METHOD SendLogMessage : BOOL
  VAR_INPUT
    str : STRING(128);
    instance : STRING(GVL_MQTT.MQTT_TOPIC_LEN) := '';
  END_VAR
                  pMqttPublishQueue^.AddMessageOn(Lane := iQueueLane,
	Payload:= CONCAT(CONCAT(instance,' | '),str),
	Topic := CONCAT(MqttDiagnosticTopic, '/Log'),
	Qos := MQTT.QoS.AtLeastOnce,
	MqttRetain := TRUE
);
                
END_METHOD

METHOD CreateSwitchEntity
  VAR_INPUT
    Name : STRING;  (* default *)
    Id : STRING;
    CommandTopic : STRING(GVL_MQTT.MQTT_TOPIC_LEN);  (* entity specific *)
    PayloadOn : STRING;
    PayloadOff : STRING;
    StateTopic : STRING(GVL_MQTT.MQTT_TOPIC_LEN);
    StateOnPayload : STRING;
    StateOffPayload : STRING;
    DeviceClass : STRING;
  END_VAR
  VAR
    EntityId : STRING(25) := 'switch';
  END_VAR
                  (* Name, id, availability and device are identical for every entity type, so
   they are filled once through the shared base struct. *)
THIS^.FillCommonFields(
	pBase := ADR(stMqttDiscMsgSwitch),
	EntityId := EntityId,
	Name := name,
	Id := Id);

// Entity related: Specific
stMqttDiscMsgSwitch.cmd_t.CharString := CommandTopic;
stMqttDiscMsgSwitch.pl_on.CharString := PayloadOn;
stMqttDiscMsgSwitch.pl_off.CharString := PayloadOff;
stMqttDiscMsgSwitch.stat_t.CharString := StateTopic;
stMqttDiscMsgSwitch.stat_on.CharString := StateOnPayload;
stMqttDiscMsgSwitch.stat_off.CharString := StateOffPayload;
stMqttDiscMsgSwitch.opt.Boolean := FALSE;
stMqttDiscMsgSwitch.dev_cla.CharString := DeviceClass;



THIS^.PublishEntityConfig(
	pStruct := ADR(stMqttDiscMsgSwitch),
	StructSize := SIZEOF(stMqttDiscMsgSwitch),
	EntityId := EntityId,
	Id := Id);
                
END_METHOD

METHOD CreateLightDimmerEntity
  VAR_INPUT
    Name : STRING;  (* default *)
    Id : STRING;
    CommandTopic : STRING(GVL_MQTT.MQTT_TOPIC_LEN);  (* entity specific *)
    PayloadOn : STRING;
    PayloadOff : STRING;
    StateTopic : STRING(GVL_MQTT.MQTT_TOPIC_LEN);
    BrightnessCommandTopic : STRING(GVL_MQTT.MQTT_TOPIC_LEN);
    BrightnessStateTopic : STRING(GVL_MQTT.MQTT_TOPIC_LEN);
    BrightnessScale : INT;
    OnCommandType : STRING := 'last';
    DmxChannel : INT := 0;  (* dmx specific *)
    DmxWidth : INT := 0;
    DmxUniverse : INT := 0;
  END_VAR
  VAR
    EntityId : STRING(25) := 'light';
  END_VAR
                  (* Name, id, availability and device are identical for every entity type, so
   they are filled once through the shared base struct. *)
THIS^.FillCommonFields(
	pBase := ADR(stMqttDiscMsgLightDim),
	EntityId := EntityId,
	Name := name,
	Id := Id);

// Entity related: Specific
stMqttDiscMsgLightDim.cmd_t.CharString := CommandTopic;
stMqttDiscMsgLightDim.pl_on.CharString := PayloadOn;
stMqttDiscMsgLightDim.pl_off.CharString := PayloadOff;
stMqttDiscMsgLightDim.stat_t.CharString := StateTopic;
stMqttDiscMsgLightDim.opt.Boolean := FALSE;

stMqttDiscMsgLightDim.bri_cmd_t.CharString := BrightnessCommandTopic;
stMqttDiscMsgLightDim.bri_stat_t.CharString := BrightnessStateTopic;
stMqttDiscMsgLightDim.bri_scl.Integer := BrightnessScale;
stMqttDiscMsgLightDim.on_cmd_type.CharString := OnCommandType;

stMqttDiscMsgLightDim.dmxChannel.Integer := DmxChannel;
stMqttDiscMsgLightDim.dmxWidth.Integer := DmxWidth;
stMqttDiscMsgLightDim.dmxUniverse.Integer := DmxUniverse;



THIS^.PublishEntityConfig(
	pStruct := ADR(stMqttDiscMsgLightDim),
	StructSize := SIZEOF(stMqttDiscMsgLightDim),
	EntityId := EntityId,
	Id := Id);
                
END_METHOD

METHOD CreateSensorEntity
  VAR_INPUT
    Name : STRING;  (* default *)
    Id : STRING;
    StateTopic : STRING(GVL_MQTT.MQTT_TOPIC_LEN);  (* entity specific *)
    ExpiryAfter : INT := 0;
    DeviceClass : STRING := '';  (* Empty publishes null, which is what Home Assistant wants for a sensor with no device class. It used to default to the string 'None', which is not a device class Home Assistant knows: it rejects the whole config and the entity never appears. Every caller passed a class, so the default was never exercised until one legitimately had none. *)
    UnitOfMeasurement : STRING := '';
    StateClass : STRING := '';  (* Home Assistant state_class: 'measurement', 'total' or 'total_increasing'. Empty publishes null, which is right for anything Home Assistant should not keep statistics on; a kWh total needs 'total_increasing' or it never reaches the energy dashboard. *)
    AvailabilityTopic : STRING(GVL_MQTT.MQTT_TOPIC_LEN) := '';  (* Overrides this entity's SECOND availability topic, so one entity can go unavailable while the rest of the device stays up. Empty keeps the device's own, which is what every other caller wants. *)
  END_VAR
  VAR
    EntityId : STRING(25) := 'sensor';
  END_VAR
                  (* Name, id, availability and device are identical for every entity type, so
   they are filled once through the shared base struct. *)
THIS^.FillCommonFields(
	pBase := ADR(stMqttDiscMsgSensor),
	EntityId := EntityId,
	Name := name,
	Id := Id);

(* One entity can be made to go unavailable on its own. The PLC's discovery
   device fills both availability slots with the same topic, so slot 2 carries
   nothing that is lost by overriding it - and avty_mode is 'all', so the entity
   is shown only while the PLC and this topic both say online. *)
IF AvailabilityTopic <> '' THEN
	stMqttDiscMsgSensor.avty[2].topic.CharString := AvailabilityTopic;
END_IF

// Entity related: Specific
//MqttDiscoverySensorMessage.ic.CharString := Icon;
stMqttDiscMsgSensor.stat_t.CharString := StateTopic;
stMqttDiscMsgSensor.exp_aft.Integer := ExpiryAfter;
(* An empty device class has to publish null rather than the empty string: Home
   Assistant validates dev_cla against a fixed list and rejects the whole config
   otherwise, which loses the entity rather than just its class. Same reason the
   unit is nulled below. *)
IF DeviceClass <> '' THEN
	stMqttDiscMsgSensor.dev_cla.CharString := DeviceClass;
ELSE
	stMqttDiscMsgSensor.dev_cla.Null := 'null';
END_IF
IF UnitOfMeasurement <> '' THEN
	stMqttDiscMsgSensor.unit_of_meas.CharString := UnitOfMeasurement;
ELSE
	stMqttDiscMsgSensor.unit_of_meas.Null := 'null';
END_IF
IF StateClass <> '' THEN
	stMqttDiscMsgSensor.stat_cla.CharString := StateClass;
ELSE
	stMqttDiscMsgSensor.stat_cla.Null := 'null';
END_IF

THIS^.PublishEntityConfig(
	pStruct := ADR(stMqttDiscMsgSensor),
	StructSize := SIZEOF(stMqttDiscMsgSensor),
	EntityId := EntityId,
	Id := Id);
                
END_METHOD

METHOD CreateSirenEntity
  VAR_INPUT
    Name : STRING;  (* default *)
    Id : STRING;
    CommandTopic : STRING(GVL_MQTT.MQTT_TOPIC_LEN);  (* entity specific *)
    PayloadOn : STRING;
    PayloadOff : STRING;
    StateTopic : STRING(GVL_MQTT.MQTT_TOPIC_LEN);
    StateOnPayload : STRING;
    StateOffPayload : STRING;
  END_VAR
  VAR
    EntityId : STRING(25) := 'siren';
  END_VAR
                  (* Name, id, availability and device are identical for every entity type, so
   they are filled once through the shared base struct. *)
THIS^.FillCommonFields(
	pBase := ADR(stMqttDiscMsgSiren),
	EntityId := EntityId,
	Name := name,
	Id := Id);

// Entity related: Specific
stMqttDiscMsgSiren.cmd_t.CharString := CommandTopic;
stMqttDiscMsgSiren.pl_on.CharString := PayloadOn;
stMqttDiscMsgSiren.pl_off.CharString := PayloadOff;
stMqttDiscMsgSiren.stat_t.CharString := StateTopic;
stMqttDiscMsgSiren.stat_on.CharString := StateOnPayload;
stMqttDiscMsgSiren.stat_off.CharString := StateOffPayload;
stMqttDiscMsgSiren.opt.Boolean := FALSE;



THIS^.PublishEntityConfig(
	pStruct := ADR(stMqttDiscMsgSiren),
	StructSize := SIZEOF(stMqttDiscMsgSiren),
	EntityId := EntityId,
	Id := Id);
                
END_METHOD

METHOD CreateLockEntity
  VAR_INPUT
    Name : STRING;  (* default *)
    Id : STRING;
    CommandTopic : STRING(GVL_MQTT.MQTT_TOPIC_LEN);  (* entity specific *)
    PayloadLock : STRING;
    PayloadUnlock : STRING;
    StateTopic : STRING(GVL_MQTT.MQTT_TOPIC_LEN);
    StateLocked : STRING;
    StateUnlocked : STRING;
  END_VAR
  VAR
    EntityId : STRING(25) := 'lock';
  END_VAR
                  (* Name, id, availability and device are identical for every entity type, so
   they are filled once through the shared base struct. *)
THIS^.FillCommonFields(
	pBase := ADR(stMqttDiscMsgLock),
	EntityId := EntityId,
	Name := name,
	Id := Id);

// Entity related: Specific
stMqttDiscMsgLock.cmd_t.CharString := CommandTopic;
stMqttDiscMsgLock.pl_lock.CharString := PayloadLock;
stMqttDiscMsgLock.pl_unlk.CharString := PayloadUnlock;
stMqttDiscMsgLock.stat_t.CharString := StateTopic;
stMqttDiscMsgLock.stat_locked.CharString := StateLocked;
stMqttDiscMsgLock.stat_unlocked.CharString := StateUnlocked;
stMqttDiscMsgLock.opt.Boolean := FALSE;



THIS^.PublishEntityConfig(
	pStruct := ADR(stMqttDiscMsgLock),
	StructSize := SIZEOF(stMqttDiscMsgLock),
	EntityId := EntityId,
	Id := Id);
                
END_METHOD

METHOD CreateLightEntity
  VAR_INPUT
    Name : STRING;  (* default *)
    Id : STRING;
    CommandTopic : STRING(GVL_MQTT.MQTT_TOPIC_LEN);  (* entity specific *)
    PayloadOn : STRING;
    PayloadOff : STRING;
    StateTopic : STRING(GVL_MQTT.MQTT_TOPIC_LEN);
  END_VAR
  VAR
    EntityId : STRING(25) := 'light';
  END_VAR
                  (* Name, id, availability and device are identical for every entity type, so
   they are filled once through the shared base struct. *)
THIS^.FillCommonFields(
	pBase := ADR(stMqttDiscMsgLight),
	EntityId := EntityId,
	Name := name,
	Id := Id);

// Entity related: Specific
stMqttDiscMsgLight.cmd_t.CharString := CommandTopic;
stMqttDiscMsgLight.pl_on.CharString := PayloadOn;
stMqttDiscMsgLight.pl_off.CharString := PayloadOff;
stMqttDiscMsgLight.stat_t.CharString := StateTopic;
stMqttDiscMsgLight.opt.Boolean := FALSE;



THIS^.PublishEntityConfig(
	pStruct := ADR(stMqttDiscMsgLight),
	StructSize := SIZEOF(stMqttDiscMsgLight),
	EntityId := EntityId,
	Id := Id);
                
END_METHOD

METHOD initBaseDevice
  VAR_INPUT
    Name : STRING;
    ConfigurationUrl : STRING := 'https://github.com/MichielVanwelsenaere/HomeAutomation.CoDeSys3';
    Identifiers : STRING;
    Manufacturer : STRING := 'unknown';
    Model : STRING := 'unknown';
    SoftwareVersion : STRING := 'unknown';
    HardwareVersion : STRING := 'unknown';
    IpAddress : STRING := '';
    MacAddress : STRING := '';
    availabilityTopic : STRING(GVL_MQTT.MQTT_TOPIC_LEN);
    availabilityTopic2 : STRING(GVL_MQTT.MQTT_TOPIC_LEN) := '';
    availabilityOnline : STRING;
    availabilityOffline : STRING;
    MqttDiscoveryPrefix : STRING;
    MqttDiagnosticTopic : STRING(GVL_MQTT.MQTT_TOPIC_LEN);
    pMqttPublishQueue : POINTER TO FB_MQTT_PUBLISH_QUEUE;
  END_VAR
                  THIS^.availabilityTopic1 := availabilityTopic;

IF CommonTypesAndFunctions.StrEquals(str1:= ADR(availabilityTopic2), str2:= ADR('')) THEN
	THIS^.availabilityTopic2 := availabilityTopic;
ELSE
	THIS^.availabilityTopic2 := availabilityTopic2;
END_IF

THIS^.availabilityOnline := availabilityOnline;
THIS^.availabilityOffline := availabilityOffline;
THIS^.pMqttPublishQueue := pMqttPublishQueue;
THIS^.MqttDiscoveryPrefix := MqttDiscoveryPrefix;
THIS^.MqttDiagnosticTopic := MqttDiagnosticTopic;

THIS^.name := Name;
THIS^.cu:= ConfigurationUrl;
THIS^.ids:= Identifiers;
THIS^.mf:= Manufacturer;
THIS^.mdl:= Model;
THIS^.hw:= HardwareVersion;
THIS^.sw:= SoftwareVersion;
THIS^.ip := IpAddress;
THIS^.sMac := MacAddress;

//Create a diagnostics availability binary sensor
CreateBinarySensorEntityWithCategory(
	Name := 'Availability',
	Id := CONCAT(Identifiers,'_diag_availability'),
	StateTopic := THIS^.availabilityTopic2,
	PayloadOn := availabilityOnline,
	PayloadOff := availabilityOffline,
	DeviceClass := 'CONNECTIVITY',
	EntityCategory := 'diagnostic');
	
//Logger
CreateDiagnosticSensorEntity(
		Name := 'Log',
		Id := CONCAT(Identifiers,'_diag_log'),
		StateTopic := CONCAT(MqttDiagnosticTopic, '/Log'));


                
END_METHOD

METHOD CreateCoverEntity
  VAR_INPUT
    Name : STRING;  (* default *)
    Id : STRING;
    CommandTopic : STRING(GVL_MQTT.MQTT_TOPIC_LEN);  (* entity specific *)
    PayloadOpen : STRING;
    PayloadClose : STRING;
    PayloadStop : STRING;
    StateTopic : STRING(GVL_MQTT.MQTT_TOPIC_LEN);
    StateOpen : STRING;
    StateOpening : STRING;
    StateClosed : STRING;
    StateClosing : STRING;
    StateStopped : STRING;
    Deviceclass : STRING;
  END_VAR
  VAR
    EntityId : STRING(25) := 'cover';
  END_VAR
                  (* Name, id, availability and device are identical for every entity type, so
   they are filled once through the shared base struct. *)
THIS^.FillCommonFields(
	pBase := ADR(stMqttDiscMsgCover),
	EntityId := EntityId,
	Name := name,
	Id := Id);

// Entity related: Specific
stMqttDiscMsgCover.cmd_t.CharString := CommandTopic;
stMqttDiscMsgCover.pl_open.CharString := PayloadOpen;
stMqttDiscMsgCover.pl_cls.CharString := PayloadClose;
stMqttDiscMsgCover.pl_stop.CharString := PayloadStop;
stMqttDiscMsgCover.stat_t.CharString := StateTopic;
stMqttDiscMsgCover.stat_open.CharString := StateOpen;
stMqttDiscMsgCover.stat_opening.CharString := StateOpening;
stMqttDiscMsgCover.stat_clsd.CharString := StateClosed;
stMqttDiscMsgCover.stat_closing.CharString := StateClosing;
stMqttDiscMsgCover.stat_stopped.CharString := StateStopped;
stMqttDiscMsgCover.opt.Boolean := FALSE;
stMqttDiscMsgCover.dev_cla.CharString := Deviceclass;



THIS^.PublishEntityConfig(
	pStruct := ADR(stMqttDiscMsgCover),
	StructSize := SIZEOF(stMqttDiscMsgCover),
	EntityId := EntityId,
	Id := Id);
                
END_METHOD

METHOD SendDeviceUpdate
  VAR_INPUT
    ConfigurationUrl : STRING := '';
    Identifiers : STRING := '';
    Manufacturer : STRING := '';
    Model : STRING := '';
    SoftwareVersion : STRING := '';
    HardwareVersion : STRING := '';
    IpAddress : STRING := '';
    MacAddress : STRING := '';
  END_VAR
  VAR
    bFoundUpdate : BOOL;
  END_VAR
                  IF ConfigurationUrl <> '' AND ConfigurationUrl <> THIS^.cu THEN 
	THIS^.cu:= ConfigurationUrl;
	bFoundUpdate := TRUE;
END_IF
IF Identifiers <> '' AND Identifiers <> THIS^.ids THEN 
	THIS^.ids:= Identifiers;
	bFoundUpdate := TRUE;
END_IF
IF Manufacturer <> '' AND Manufacturer <> THIS^.mf THEN  
	THIS^.mf:= Manufacturer;
	bFoundUpdate := TRUE;
END_IF
IF Model <> '' AND Model <> THIS^.mdl THEN  
	THIS^.mdl:= Model;
	bFoundUpdate := TRUE;
END_IF
IF HardwareVersion <> '' AND HardwareVersion <> THIS^.hw THEN  
	THIS^.hw:= HardwareVersion;
	bFoundUpdate := TRUE;
END_IF
IF SoftwareVersion <> '' AND SoftwareVersion <> THIS^.sw THEN  
	THIS^.sw:= SoftwareVersion;
	bFoundUpdate := TRUE;
END_IF
IF IpAddress <> '' AND IpAddress <> THIS^.ip THEN  
	THIS^.ip := IpAddress;
	bFoundUpdate := TRUE;
END_IF
IF MacAddress <> '' AND MacAddress <> THIS^.sMac THEN  
	THIS^.sMac := MacAddress;
	bFoundUpdate := TRUE;
END_IF

IF bFoundUpdate THEN
	//Dummy publish just to update device description
	CreateBinarySensorEntityWithCategory(
		Name := 'Availability',
		Id := CONCAT(ids,'_diag_availability'),
		StateTopic := availabilityTopic2,
		PayloadOn := availabilityOnline,
		PayloadOff := availabilityOffline,
		DeviceClass := 'CONNECTIVITY',
		EntityCategory := 'diagnostic');	
END_IF
                
END_METHOD

{attribute 'reflection'}
METHOD CreateBinarySensorEntity
  VAR_INPUT
    Name : STRING;  (* default *)
    Id : STRING;
    StateTopic : STRING(GVL_MQTT.MQTT_TOPIC_LEN);  (* entity specific *)
    PayloadOn : STRING;
    PayloadOff : STRING;
    DeviceClass : STRING;
  END_VAR
  VAR
    EntityId : STRING(25) := 'binary_sensor';
  END_VAR
                  (* Name, id, availability and device are identical for every entity type, so
   they are filled once through the shared base struct. *)
THIS^.FillCommonFields(
	pBase := ADR(stMqttDiscMsgBinSens),
	EntityId := EntityId,
	Name := name,
	Id := Id);

// Entity related: Specific
stMqttDiscMsgBinSens.stat_t.CharString := StateTopic;
stMqttDiscMsgBinSens.pl_on.CharString := PayloadOn;
stMqttDiscMsgBinSens.pl_off.CharString := PayloadOff;
stMqttDiscMsgBinSens.dev_cla.CharString := DeviceClass;



THIS^.PublishEntityConfig(
	pStruct := ADR(stMqttDiscMsgBinSens),
	StructSize := SIZEOF(stMqttDiscMsgBinSens),
	EntityId := EntityId,
	Id := Id);
                
END_METHOD

{attribute 'reflection'}
METHOD CreateBinarySensorEntityWithCategory
  VAR_INPUT
    Name : STRING;  (* default *)
    Id : STRING;
    StateTopic : STRING(GVL_MQTT.MQTT_TOPIC_LEN);  (* entity specific *)
    PayloadOn : STRING;
    PayloadOff : STRING;
    DeviceClass : STRING;
    EntityCategory : STRING;  (* config or diagnostic *)
  END_VAR
  VAR
    EntityId : STRING(25) := 'binary_sensor';
  END_VAR
                  (* Name, id, availability and device are identical for every entity type, so
   they are filled once through the shared base struct. *)
THIS^.FillCommonFields(
	pBase := ADR(stMqttDiscMsgBinSensWCat),
	EntityId := EntityId,
	Name := name,
	Id := Id);

// Entity related: Specific
stMqttDiscMsgBinSensWCat.stat_t.CharString := StateTopic;
stMqttDiscMsgBinSensWCat.pl_on.CharString := PayloadOn;
stMqttDiscMsgBinSensWCat.pl_off.CharString := PayloadOff;
stMqttDiscMsgBinSensWCat.dev_cla.CharString := DeviceClass;
stMqttDiscMsgBinSensWCat.ent_cat.CharString := EntityCategory;



THIS^.PublishEntityConfig(
	pStruct := ADR(stMqttDiscMsgBinSensWCat),
	StructSize := SIZEOF(stMqttDiscMsgBinSensWCat),
	EntityId := EntityId,
	Id := Id);
                
END_METHOD

METHOD CreateEventEntity
  VAR_INPUT
    Name : STRING;  (* default *)
    Id : STRING;
    StateTopic : STRING(GVL_MQTT.MQTT_TOPIC_LEN);  (* entity specific *)
    EventTypes : ARRAY[1..3] OF STRING;
    Deviceclass : STRING;
  END_VAR
  VAR
    EntityId : STRING(25) := 'event';
  END_VAR
                  (* Name, id, availability and device are identical for every entity type, so
   they are filled once through the shared base struct. *)
THIS^.FillCommonFields(
	pBase := ADR(stMqttDiscMsgEvent),
	EntityId := EntityId,
	Name := name,
	Id := Id);

// Entity related: Specific
stMqttDiscMsgEvent.stat_t.CharString := StateTopic;
stMqttDiscMsgEvent.evt_typ[1].CharString := EventTypes[1];
stMqttDiscMsgEvent.evt_typ[2].CharString := EventTypes[2];
stMqttDiscMsgEvent.evt_typ[3].CharString := EventTypes[3];
stMqttDiscMsgEvent.dev_cla.CharString := Deviceclass;



THIS^.PublishEntityConfig(
	pStruct := ADR(stMqttDiscMsgEvent),
	StructSize := SIZEOF(stMqttDiscMsgEvent),
	EntityId := EntityId,
	Id := Id);
                
END_METHOD

METHOD CreateValveEntity
  VAR_INPUT
    Name : STRING;  (* default *)
    Id : STRING;
    CommandTopic : STRING(GVL_MQTT.MQTT_TOPIC_LEN);  (* entity specific *)
    PayloadOpen : STRING;
    PayloadClosed : STRING;
    StateTopic : STRING(GVL_MQTT.MQTT_TOPIC_LEN);
    StateOpen : STRING;
    StateClosed : STRING;
    Deviceclass : STRING;
  END_VAR
  VAR
    EntityId : STRING(25) := 'valve';
  END_VAR
                  (* Name, id, availability and device are identical for every entity type, so
   they are filled once through the shared base struct. *)
THIS^.FillCommonFields(
	pBase := ADR(stMqttDiscMsgValve),
	EntityId := EntityId,
	Name := name,
	Id := Id);

// Entity related: Specific
stMqttDiscMsgValve.cmd_t.CharString := CommandTopic;
stMqttDiscMsgValve.pl_open.CharString := PayloadOpen;
stMqttDiscMsgValve.pl_cls.CharString := PayLoadClosed;
stMqttDiscMsgValve.stat_t.CharString := StateTopic;
stMqttDiscMsgValve.stat_open.CharString := StateOpen;
stMqttDiscMsgValve.stat_clsd.CharString := StateClosed;
stMqttDiscMsgValve.opt.Boolean := FALSE;
stMqttDiscMsgValve.dev_cla.CharString := Deviceclass;



THIS^.PublishEntityConfig(
	pStruct := ADR(stMqttDiscMsgValve),
	StructSize := SIZEOF(stMqttDiscMsgValve),
	EntityId := EntityId,
	Id := Id);
                
END_METHOD

METHOD CreateClimateEntity
  VAR_INPUT
    Name : STRING;  (* default *)
    Id : STRING;
    InitialDesiredTemperature : INT;  (* entity specific *)
    CurrentTemperatureTopic : STRING(GVL_MQTT.MQTT_TOPIC_LEN);
    CurrentHumidityTopic : STRING(GVL_MQTT.MQTT_TOPIC_LEN);
    ModeCommandTopic : STRING(GVL_MQTT.MQTT_TOPIC_LEN);
    ModeStateTopic : STRING(GVL_MQTT.MQTT_TOPIC_LEN);
    TemperatureCommandTopic : STRING(GVL_MQTT.MQTT_TOPIC_LEN);
    TemperatureStateTopic : STRING(GVL_MQTT.MQTT_TOPIC_LEN);
    TempStep : REAL;
  END_VAR
  VAR
    EntityId : STRING(25) := 'climate';
  END_VAR
                  (* Name, id, availability and device are identical for every entity type, so
   they are filled once through the shared base struct. *)
THIS^.FillCommonFields(
	pBase := ADR(stMqttDiscMsgClimate),
	EntityId := EntityId,
	Name := name,
	Id := Id);

// Entity related: Specific
stMqttDiscMsgClimate.init.Integer := InitialDesiredTemperature;
stMqttDiscMsgClimate.curr_temp_t.CharString := CurrentTemperatureTopic;
stMqttDiscMsgClimate.curr_hum_t.CharString := CurrentHumidityTopic;
stMqttDiscMsgClimate.modes[1].CharString := 'auto';
stMqttDiscMsgClimate.modes[2].CharString := 'off';
stMqttDiscMsgClimate.modes[3].CharString := 'heat';
stMqttDiscMsgClimate.mode_cmd_t.CharString := ModeCommandTopic;
stMqttDiscMsgClimate.mode_stat_t.CharString := ModeStateTopic;
stMqttDiscMsgClimate.temp_cmd_t.CharString := TemperatureCommandTopic;
stMqttDiscMsgClimate.temp_stat_t.CharString := TemperatureStateTopic;
stMqttDiscMsgClimate.temp_step.Number := TempStep;
stMqttDiscMsgClimate.opt.Boolean := FALSE;



THIS^.PublishEntityConfig(
	pStruct := ADR(stMqttDiscMsgClimate),
	StructSize := SIZEOF(stMqttDiscMsgClimate),
	EntityId := EntityId,
	Id := Id);
                
END_METHOD

METHOD CreateValveStateEntity
  VAR_INPUT
    Name : STRING;  (* default *)
    Id : STRING;
    StateTopic : STRING(GVL_MQTT.MQTT_TOPIC_LEN);  (* entity specific *)
    StateOpen : STRING;
    StateClosed : STRING;
    Deviceclass : STRING;
  END_VAR
  VAR
    EntityId : STRING(25) := 'valve';
  END_VAR
                  (* Name, id, availability and device are identical for every entity type, so
   they are filled once through the shared base struct. *)
THIS^.FillCommonFields(
	pBase := ADR(stMqttDiscMsgValveState),
	EntityId := EntityId,
	Name := name,
	Id := Id);

// Entity related: Specific
stMqttDiscMsgValveState.stat_t.CharString := StateTopic;
stMqttDiscMsgValveState.stat_open.CharString := StateOpen;
stMqttDiscMsgValveState.stat_clsd.CharString := StateClosed;
stMqttDiscMsgValveState.opt.Boolean := FALSE;
stMqttDiscMsgValveState.dev_cla.CharString := Deviceclass;



THIS^.PublishEntityConfig(
	pStruct := ADR(stMqttDiscMsgValveState),
	StructSize := SIZEOF(stMqttDiscMsgValveState),
	EntityId := EntityId,
	Id := Id);
                
END_METHOD

METHOD CreateFanEntity
  VAR_INPUT
    Name : STRING;  (* default *)
    Id : STRING;
    CommandTopic : STRING(GVL_MQTT.MQTT_TOPIC_LEN);  (* entity specific - command_topic is the only key Home Assistant requires *)
    PayloadOn : STRING;
    PayloadOff : STRING;
    StateTopic : STRING(GVL_MQTT.MQTT_TOPIC_LEN);
    PercentageCommandTopic : STRING(GVL_MQTT.MQTT_TOPIC_LEN) := '';  (* speed as a percentage; leave PercentageCommandTopic empty for an on/off fan *)
    PercentageStateTopic : STRING(GVL_MQTT.MQTT_TOPIC_LEN) := '';
    SpeedRangeMin : INT := 1;
    SpeedRangeMax : INT := 100;
    OscillationCommandTopic : STRING(GVL_MQTT.MQTT_TOPIC_LEN) := '';  (* oscillation; leave OscillationCommandTopic empty to omit it *)
    OscillationStateTopic : STRING(GVL_MQTT.MQTT_TOPIC_LEN) := '';
  END_VAR
  VAR
    EntityId : STRING(25) := 'fan';
  END_VAR
                  (* Name, id, availability and device are identical for every entity type, so
   they are filled once through the shared base struct. *)
THIS^.FillCommonFields(
	pBase := ADR(stMqttDiscMsgFan),
	EntityId := EntityId,
	Name := name,
	Id := Id);

// Entity related: Specific
// command_topic is the only key Home Assistant requires for a fan.
stMqttDiscMsgFan.cmd_t.CharString := CommandTopic;
stMqttDiscMsgFan.pl_on.CharString := PayloadOn;
stMqttDiscMsgFan.pl_off.CharString := PayloadOff;
stMqttDiscMsgFan.stat_t.CharString := StateTopic;
stMqttDiscMsgFan.opt.Boolean := FALSE;

// Speed, as a percentage. Left out of the published JSON when no topic is given,
// which is what makes this an on/off-only fan.
IF NOT CommonTypesAndFunctions.StrEquals(str1:= ADR(PercentageCommandTopic), str2:= ADR('')) THEN
	stMqttDiscMsgFan.pct_cmd_t.CharString := PercentageCommandTopic;
	stMqttDiscMsgFan.pct_stat_t.CharString := PercentageStateTopic;
	stMqttDiscMsgFan.spd_rng_min.Integer := SpeedRangeMin;
	stMqttDiscMsgFan.spd_rng_max.Integer := SpeedRangeMax;
END_IF

// Oscillation, likewise optional.
IF NOT CommonTypesAndFunctions.StrEquals(str1:= ADR(OscillationCommandTopic), str2:= ADR('')) THEN
	stMqttDiscMsgFan.osc_cmd_t.CharString := OscillationCommandTopic;
	stMqttDiscMsgFan.osc_stat_t.CharString := OscillationStateTopic;
	stMqttDiscMsgFan.pl_osc_on.CharString := 'oscillate_on';
	stMqttDiscMsgFan.pl_osc_off.CharString := 'oscillate_off';
END_IF



THIS^.PublishEntityConfig(
	pStruct := ADR(stMqttDiscMsgFan),
	StructSize := SIZEOF(stMqttDiscMsgFan),
	EntityId := EntityId,
	Id := Id);
                
END_METHOD

(* Fills the part of a discovery config that is identical for every entity type. Every MQTT_DISCOVERY_* struct EXTENDS MQTT_DISCOVERY_BASE, so one pointer reaches the shared fields of all of them. *)
METHOD FillCommonFields
  VAR_INPUT
    pBase : POINTER TO MQTT_DISCOVERY_BASE;  (* ADR() of the concrete discovery struct; its base part is what gets written. *)
    EntityId : STRING(25);  (* Home Assistant platform, e.g. 'light' - used to build default_entity_id. *)
    Name : STRING;
    Id : STRING;
  END_VAR
                  IF pBase = 0 THEN
	RETURN;
END_IF

// 	Entity related: Basis
pBase^.name.CharString :=  Name; // friendly name
pBase^.default_entity_id.CharString :=  CONCAT(CONCAT(EntityId, '.'), Id);
pBase^.uniq_id.CharString :=  Id;

// Availabilty related
pBase^.avty[1].topic.CharString := THIS^.availabilityTopic1;
pBase^.avty[2].topic.CharString := THIS^.availabilityTopic2;
pBase^.avty_mode.CharString := 'all';
pBase^.pl_avail.CharString :=   THIS^.availabilityOnline;
pBase^.pl_not_avail.CharString :=  THIS^.availabilityOffline;
pBase^.qos.Integer := 2;

// Device related
pBase^.dev.cu.CharString := THIS^.cu;
pBase^.dev.name.CharString := THIS^.name;
pBase^.dev.hw.CharString := THIS^.hw;
pBase^.dev.ids.CharString := THIS^.ids;
pBase^.dev.sw.CharString := THIS^.sw;
pBase^.dev.mdl.CharString := THIS^.mdl;
pBase^.dev.mf.CharString := THIS^.mf;

                
END_METHOD

(* Composes the discovery JSON for an already-filled struct and publishes it to the entity's config topic. Returns TRUE when a payload was queued. *)
METHOD PublishEntityConfig : BOOL
  VAR_INPUT
    pStruct : POINTER TO BYTE;  (* ADR() of the concrete discovery struct. *)
    StructSize : UDINT;  (* SIZEOF() of that same struct - the caller must pass it, because this method only sees a pointer and SIZEOF here would measure the pointer. *)
    EntityId : STRING(25);
    Id : STRING;
  END_VAR
  VAR
    fbComposeJSON : STRUCT_TO_JSON;
    sMqttJSON : STRING(1500);
    sMqttTopic : STRING(GVL_MQTT.MQTT_TOPIC_LEN);
    bStripJsonRootOk : BOOL;
    bJsonComplete : BOOL;
    pJsonByte : POINTER TO BYTE;  (* Used to find where sMqttJSON really ends. A pointer walk, not RIGHT() or LEN(): those are declared over STRING(255) and narrow a longer argument without saying so. See the comment in the body. *)
    diJsonLen : DINT;
    diI : DINT;
    bKeyRenamed : BOOL;  (* Result of a key rename. Nothing acts on it: a config with no such key is the ordinary case, and the truncation guard below catches anything that did go wrong far more reliably than this flag would. *)
  END_VAR
                  PublishEntityConfig := FALSE;
IF pStruct = 0 OR StructSize = 0 THEN
	RETURN;
END_IF

sMqttTopic := CONCAT(CONCAT(CONCAT(CONCAT(THIS^.MqttDiscoveryPrefix, EntityId),'/'), Id),'/config' );

fbComposeJSON(
	JSONString:= ADR(sMqttJSON),
	JSONStringSize:= SIZEOF(sMqttJSON),
	JSONVars:= pStruct,
	NumberOfVars:= StructSize / SIZEOF(JSONVAR),
	MaxLevel := 3,
	Rootless := TRUE,
);
fbComposeJSON.Execute := TRUE;
fbComposeJSON();

bStripJsonRootOk := F_STRIP_JSON_ROOT(pJson := ADR(sMqttJSON), uiSize := SIZEOF(sMqttJSON));

(* A few Home Assistant keys are IEC operators, so no struct can declare them
   under the name they have to be published as. A number entity needs min and
   max; the struct carries min_val and max_val, and they are corrected here.

   Done for every entity type rather than only for numbers: the scan is over a
   config that has already been composed, it runs at the handful of publishes
   that happen at startup, and a config containing neither key costs one failed
   search. Putting it here means the next struct that hits the same collision
   needs no new plumbing. *)
bKeyRenamed := F_JSON_RENAME_KEY(pJson := ADR(sMqttJSON), uiSize := SIZEOF(sMqttJSON),
							sFrom := '"min_val"', sTo := '"min"');
bKeyRenamed := F_JSON_RENAME_KEY(pJson := ADR(sMqttJSON), uiSize := SIZEOF(sMqttJSON),
							sFrom := '"max_val"', sTo := '"max"');

(* A composed config that does not end in a closing brace is truncated, and
   publishing it is worse than publishing nothing: Home Assistant rejects the
   whole config and the entity silently disappears, while the log cheerfully
   reports the discovery as added.

   Walk to the null terminator rather than asking a string function where the
   end is. This check used to read

       bJsonComplete := RIGHT(sMqttJSON, 1) = '}';

   and RIGHT is declared over STRING(255), so sMqttJSON was silently narrowed to
   its first 255 bytes on the way in and RIGHT returned character 255 instead of
   the last one. Every discovery config here is longer than that, so the guard
   rejected all of them - and this PLC published no discovery config at all
   between that check landing and this fix. The buffer was never the problem:
   1500 bytes with 665 in use. The FUNCTION SIGNATURE was the narrow part, in a
   check whose whole job is detecting values that got cut short. *)
pJsonByte := ADR(sMqttJSON);
diJsonLen := 0;
FOR diI := 0 TO UDINT_TO_DINT(SIZEOF(sMqttJSON)) - 1 DO
	IF pJsonByte[diI] = 0 THEN
		diJsonLen := diI;
		EXIT;
	END_IF
END_FOR
bJsonComplete := (diJsonLen > 0) AND (pJsonByte[diJsonLen - 1] = 16#7D);

IF sMqttJSON = '' THEN
	SendLogMessage(str:=CONCAT(CONCAT('ERROR ',Id), ' had empty MqttJSON'), instance := sInstanceName);
ELSIF bStripJsonRootOk = FALSE THEN
	SendLogMessage(str:=CONCAT(CONCAT('ERROR ',Id), ' failed json root strip'), instance := sInstanceName);
ELSIF NOT bJsonComplete THEN
	SendLogMessage(str:=CONCAT(CONCAT('ERROR ',Id), ' composed truncated json'), instance := sInstanceName);
ELSIF NOT (sMqttJSON = '') THEN
	pMqttPublishQueue^.AddMessageOn(Lane := iQueueLane,
		Payload:= sMqttJSON,
		Topic := sMqttTopic,
		Qos := MQTT.QoS.ExactlyOnce,
		MqttRetain := TRUE,
	);
	SendLogMessage(str:=CONCAT(CONCAT('Added ',Id), ' as MQTT discovery'), instance := sInstanceName);
	PublishEntityConfig := TRUE;
END_IF
                
END_METHOD

METHOD CreateCoverEntityWithPosition
  VAR_INPUT
    Name : STRING;  (* default *)
    Id : STRING;
    CommandTopic : STRING(GVL_MQTT.MQTT_TOPIC_LEN);  (* entity specific *)
    PayloadOpen : STRING;
    PayloadClose : STRING;
    PayloadStop : STRING;
    StateTopic : STRING(GVL_MQTT.MQTT_TOPIC_LEN);
    StateOpen : STRING;
    StateOpening : STRING;
    StateClosed : STRING;
    StateClosing : STRING;
    StateStopped : STRING;
    Deviceclass : STRING;
    PositionTopic : STRING(GVL_MQTT.MQTT_TOPIC_LEN);  (* Where the cover reports how far open it is. *)
    SetPositionTopic : STRING(GVL_MQTT.MQTT_TOPIC_LEN);  (* Where Home Assistant asks for a position. **Supplying this is what puts a slider on the entity** rather than three buttons. *)
    PositionOpen : INT := 100;  (* The numbers that mean fully open and fully closed. Home Assistant's own defaults, and there is no good reason to differ - a cover that counts some other way should convert before publishing rather than teach every reader a private scale. *)
    PositionClosed : INT := 0;
  END_VAR
  VAR
    EntityId : STRING(25) := 'cover';
  END_VAR
                  (* A cover with a position slider, published from its own struct.

   Deliberately a second method and a second struct rather than four optional
   parameters on CreateCoverEntity, because Home Assistant will not accept the
   fields as null. It validates set_position_topic and position_topic as strings,
   and a null fails the whole config rather than just the slider:

     Error 'string value is None for dictionary value @ data['set_position_topic']'
     when processing MQTT discovery message topic:
     'homeassistant/cover/..._FB_DO_COVER_001/config'

   which cost a working cover entity for as long as the null was published. A key
   that must not be there cannot be nulled; it has to be absent, and the way this
   project makes a key absent is a struct without it. Same reason
   MQTT_DISCOVERY_BINARY_SENSOR_ENT_CAT exists beside MQTT_DISCOVERY_BINARY_SENSOR
   rather than the category being an optional field. *)
THIS^.FillCommonFields(
	pBase := ADR(stMqttDiscMsgCoverPos),
	EntityId := EntityId,
	Name := name,
	Id := Id);

// Entity related: Specific
stMqttDiscMsgCoverPos.cmd_t.CharString := CommandTopic;
stMqttDiscMsgCoverPos.pl_open.CharString := PayloadOpen;
stMqttDiscMsgCoverPos.pl_cls.CharString := PayloadClose;
stMqttDiscMsgCoverPos.pl_stop.CharString := PayloadStop;
stMqttDiscMsgCoverPos.stat_t.CharString := StateTopic;
stMqttDiscMsgCoverPos.stat_open.CharString := StateOpen;
stMqttDiscMsgCoverPos.stat_opening.CharString := StateOpening;
stMqttDiscMsgCoverPos.stat_clsd.CharString := StateClosed;
stMqttDiscMsgCoverPos.stat_closing.CharString := StateClosing;
stMqttDiscMsgCoverPos.stat_stopped.CharString := StateStopped;
stMqttDiscMsgCoverPos.opt.Boolean := FALSE;
stMqttDiscMsgCoverPos.dev_cla.CharString := Deviceclass;

// Position
stMqttDiscMsgCoverPos.pos_t.CharString := PositionTopic;
stMqttDiscMsgCoverPos.set_pos_t.CharString := SetPositionTopic;
stMqttDiscMsgCoverPos.pos_open.Integer := PositionOpen;
stMqttDiscMsgCoverPos.pos_clsd.Integer := PositionClosed;

THIS^.PublishEntityConfig(
	pStruct := ADR(stMqttDiscMsgCoverPos),
	StructSize := SIZEOF(stMqttDiscMsgCoverPos),
	EntityId := EntityId,
	Id := Id);
                
END_METHOD

(* Announce a Home Assistant number: a value somebody can set, with a range and a step, and a state topic carrying what the device actually holds. *)
METHOD CreateNumberEntity
  VAR_INPUT
    Name : STRING;
    Id : STRING;
    CommandTopic : STRING(GVL_MQTT.MQTT_TOPIC_LEN);
    StateTopic : STRING(GVL_MQTT.MQTT_TOPIC_LEN);  (* Where the value the device actually holds is published. Leave empty only if the register genuinely cannot be read back. *)
    MinValue : INT;  (* Signed: a release-the-override value of -1 is a real setting on some devices. *)
    MaxValue : INT;
    StepValue : INT;
    UnitOfMeasurement : STRING;
    DeviceClass : STRING;
    EntityCategory : STRING;  (* 'config' keeps a setpoint off the main dashboard. Empty for none. *)
    SliderMode : BOOL;  (* TRUE for a slider, FALSE for a typed box. *)
  END_VAR
  VAR
    EntityId : STRING(25) := 'number';
  END_VAR
                  (* Name, id, availability and device are identical for every entity type, so
   they are filled once through the shared base struct. *)
THIS^.FillCommonFields(
	pBase := ADR(stMqttDiscMsgNumber),
	EntityId := EntityId,
	Name := Name,
	Id := Id);

// Entity related: Specific
stMqttDiscMsgNumber.cmd_t.CharString := CommandTopic;
stMqttDiscMsgNumber.stat_t.CharString := StateTopic;
(* min_val / max_val, not min / max: MIN and MAX are IEC operators and cannot
   be member names, and PRO_JSON takes the JSON key from the member name -
   JSONVAR has no name field to override it. PublishEntityConfig renames both
   keys on the way out, because Home Assistant accepts only min and max. *)
stMqttDiscMsgNumber.min_val.Integer := MinValue;
stMqttDiscMsgNumber.max_val.Integer := MaxValue;
stMqttDiscMsgNumber.step.Integer := StepValue;
(* Empty means absent, and absent has to be published as null rather than an
   empty string: Home Assistant validates these against fixed lists and
   rejects the entire config when one does not match, so the entity is lost
   rather than just its class. CreateSensorEntity does the same. *)
IF UnitOfMeasurement <> '' THEN
	stMqttDiscMsgNumber.unit_of_meas.CharString := UnitOfMeasurement;
ELSE
	stMqttDiscMsgNumber.unit_of_meas.Null := 'null';
END_IF
IF DeviceClass <> '' THEN
	stMqttDiscMsgNumber.dev_cla.CharString := DeviceClass;
ELSE
	stMqttDiscMsgNumber.dev_cla.Null := 'null';
END_IF
IF EntityCategory <> '' THEN
	stMqttDiscMsgNumber.ent_cat.CharString := EntityCategory;
ELSE
	stMqttDiscMsgNumber.ent_cat.Null := 'null';
END_IF

(* A slider cannot be aimed at 800 ppm in steps of 10, and a typed box is
   tedious for a 0-100 percentage. Only the caller knows the range, so only the
   caller can choose. *)
IF SliderMode THEN
	stMqttDiscMsgNumber.mode.CharString := 'slider';
ELSE
	stMqttDiscMsgNumber.mode.CharString := 'box';
END_IF

(* Never optimistic. Every number this project announces sits on a register that
   can be read back, so Home Assistant shows what the device holds rather than
   what somebody last sent it - which matters when the same setting is also
   changeable from a wall control. *)
stMqttDiscMsgNumber.opt.Boolean := FALSE;

THIS^.PublishEntityConfig(
	pStruct := ADR(stMqttDiscMsgNumber),
	StructSize := SIZEOF(stMqttDiscMsgNumber),
	EntityId := EntityId,
	Id := Id);
                
END_METHOD

(* Announce a Home Assistant button: a stateless command. Right wherever the device has an action but nothing readable that reports it back. *)
METHOD CreateButtonEntity
  VAR_INPUT
    Name : STRING;
    Id : STRING;
    CommandTopic : STRING(GVL_MQTT.MQTT_TOPIC_LEN);
    PayloadPress : STRING;  (* What is sent on press. *)
    EntityCategory : STRING;  (* 'config' or 'diagnostic'. Empty for none. *)
    DeviceClass : STRING;  (* Only identify, restart and update exist for a button. Usually empty. *)
  END_VAR
  VAR
    EntityId : STRING(25) := 'button';
  END_VAR
                  (* Name, id, availability and device are identical for every entity type, so
   they are filled once through the shared base struct. *)
THIS^.FillCommonFields(
	pBase := ADR(stMqttDiscMsgButton),
	EntityId := EntityId,
	Name := Name,
	Id := Id);

// Entity related: Specific
stMqttDiscMsgButton.cmd_t.CharString := CommandTopic;
stMqttDiscMsgButton.pl_prs.CharString := PayloadPress;
(* Empty means absent, and absent has to be published as null rather than an
   empty string: Home Assistant validates these against fixed lists and
   rejects the entire config when one does not match, so the entity is lost
   rather than just its class. CreateSensorEntity does the same. *)
IF EntityCategory <> '' THEN
	stMqttDiscMsgButton.ent_cat.CharString := EntityCategory;
ELSE
	stMqttDiscMsgButton.ent_cat.Null := 'null';
END_IF
IF DeviceClass <> '' THEN
	stMqttDiscMsgButton.dev_cla.CharString := DeviceClass;
ELSE
	stMqttDiscMsgButton.dev_cla.Null := 'null';
END_IF

(* No state topic and no optimistic flag: a button has no state to be right or
   wrong about. Where the result IS observable, the thing wanted is a select or
   a number, not a button. *)

THIS^.PublishEntityConfig(
	pStruct := ADR(stMqttDiscMsgButton),
	StructSize := SIZEOF(stMqttDiscMsgButton),
	EntityId := EntityId,
	Id := Id);
                
END_METHOD

(* Put this device's publishes on a given queue lane. Call once, after init, from the block that owns it - and only with the lane of the task it runs in. *)
METHOD SetLane
  VAR_INPUT
    Lane : INT;
  END_VAR
                  THIS^.iQueueLane := Lane;

                
END_METHOD
END_FUNCTION_BLOCK

FUNCTION_BLOCK FB_DFROBOT_MQTT_DISCOVERY_DEVICE EXTENDS FB_BASE_MQTT_DISCOVERY_DEVICE
  VAR
    Manufacturer : STRING := 'DFRobot';  (* Fixed for this block - every sensor it serves is a DFRobot one. The model varies (SEN0492 today, and the rest of the RS485 range would fit here), so it is passed in per instance instead. Same shape as FB_EASTRON_SDM_MQTT_DISCOVERY_DEVICE. *)
  END_VAR

            
          

METHOD initDFRobotDevice
  VAR_INPUT
    name : STRING;
    id : STRING;
    Model : STRING := 'unknown';  (* Model shown on the Home Assistant device page. One discovery device serves the whole DFRobot RS485 range, so the model is set per instance. *)
    availabilityTopic1 : STRING(GVL_MQTT.MQTT_TOPIC_LEN);
    availabilityTopic2 : STRING(GVL_MQTT.MQTT_TOPIC_LEN) := '';
    availabilityOnline : STRING;
    availabilityOffline : STRING;
    MqttDiscoveryPrefix : STRING;
    MqttDiagnosticTopic : STRING(GVL_MQTT.MQTT_TOPIC_LEN);
    pMqttPublishQueue : POINTER TO FB_MQTT_PUBLISH_QUEUE;
  END_VAR
                  (* Announces the sensor itself as a Home Assistant device, so its measurements
   group under one card instead of scattering across the PLC device. *)
IF bInit THEN
	bInit := FALSE;

	SUPER^.initBaseDevice(
		Name := name,
		Identifiers := id,
		Manufacturer := THIS^.Manufacturer,
		Model := Model,
		availabilityTopic := availabilityTopic1,
		availabilityTopic2 := availabilityTopic2,
		availabilityOnline := availabilityOnline,
		availabilityOffline := availabilityOffline,
		MqttDiscoveryPrefix := MqttDiscoveryPrefix,
		MqttDiagnosticTopic := MqttDiagnosticTopic,
		pMqttPublishQueue := pMqttPublishQueue);
END_IF

                
END_METHOD
END_FUNCTION_BLOCK

FUNCTION_BLOCK FB_EASTRON_SDM_MQTT_DISCOVERY_DEVICE EXTENDS FB_BASE_MQTT_DISCOVERY_DEVICE
  VAR
    Manufacturer : STRING := 'Eastron';  (* Fixed for this block - every SDM is an Eastron meter. The model varies (SDM120, SDM220, SDM630), so it is passed in per instance instead. *)
  END_VAR

            
          

METHOD initEastronDevice
  VAR_INPUT
    name : STRING;
    id : STRING;
    Model : STRING := 'unknown';
    availabilityTopic1 : STRING(GVL_MQTT.MQTT_TOPIC_LEN);
    availabilityTopic2 : STRING(GVL_MQTT.MQTT_TOPIC_LEN) := '';
    availabilityOnline : STRING;
    availabilityOffline : STRING;
    MqttDiscoveryPrefix : STRING;
    MqttDiagnosticTopic : STRING(GVL_MQTT.MQTT_TOPIC_LEN);
    pMqttPublishQueue : POINTER TO FB_MQTT_PUBLISH_QUEUE;
  END_VAR
                  (* Announces the meter itself as a Home Assistant device, so its measurements
   group under one card instead of scattering across the PLC device. Same shape
   as FB_1WIRE_MQTT_DISCOVERY_DEVICE, with Model passed through because one
   block serves the whole SDM family. *)
IF bInit THEN
	bInit := FALSE;

	SUPER^.initBaseDevice(
		Name := name,
		Identifiers := id,
		Manufacturer := THIS^.Manufacturer,
		Model := Model,
		availabilityTopic := availabilityTopic1,
		availabilityTopic2 := availabilityTopic2,
		availabilityOnline := availabilityOnline,
		availabilityOffline := availabilityOffline,
		MqttDiscoveryPrefix := MqttDiscoveryPrefix,
		MqttDiagnosticTopic := MqttDiagnosticTopic,
		pMqttPublishQueue := pMqttPublishQueue);
END_IF
                
END_METHOD
END_FUNCTION_BLOCK

{attribute 'reflection'}
FUNCTION_BLOCK FB_PLC_MQTT_DISCOVERY_DEVICE EXTENDS FB_BASE_MQTT_DISCOVERY_DEVICE

            
          

(* FB_Init is always available implicitly and it is used primarily for initialization. The return value is not evaluated. For a specific influence, you can also declare the methods explicitly and provide additional code there with the standard initialization code. You can evaluate the return value. *)
METHOD FB_init : BOOL
  VAR_INPUT
    bInitRetains : BOOL;  (* TRUE: the retain variables are initialized (reset warm / reset cold) *)
    bInCopyCode : BOOL;  (* TRUE: the instance will be copied to the copy code afterward (online change) *)
    friendlyName : STRING;
    id : STRING;
    manufacturer : STRING;
    availabilityTopic : STRING(GVL_MQTT.MQTT_TOPIC_LEN);
    availabilityOnline : STRING;
    availabilityOffline : STRING;
    MqttDiscoveryPrefix : STRING;
    MqttDiagnosticTopic : STRING(GVL_MQTT.MQTT_TOPIC_LEN);
    pMqttPublishQueue : POINTER TO FB_MQTT_PUBLISH_QUEUE;
  END_VAR
                  IF bInit THEN
    bInit := FALSE;
	
	SUPER^.initBaseDevice(
		Name := friendlyName,
		Identifiers := id,
		Manufacturer := manufacturer,
		availabilityTopic := availabilityTopic,
		availabilityTopic2 := availabilityTopic,			
		availabilityOnline := availabilityOnline,
		availabilityOffline := availabilityOffline,
		MqttDiscoveryPrefix := MqttDiscoveryPrefix,
		MqttDiagnosticTopic := MqttDiagnosticTopic,
		pMqttPublishQueue := pMqttPublishQueue);
END_IF
                
END_METHOD
END_FUNCTION_BLOCK

FUNCTION F_SWAP_WORDS_TO_REAL : REAL
  VAR_INPUT
    wHi : WORD;
    wLo : WORD;
  END_VAR
  VAR
    dwVar : DWORD;
    prReal : POINTER TO REAL;
  END_VAR

            dwVar := SHL(WORD_TO_DWORD(wHi),16) OR WORD_TO_DWORD(wLo);
prReal := ADR(dwVar);
F_SWAP_WORDS_TO_REAL := prReal^;
          
END_FUNCTION

(* Arbitrates one RS485 bus between the aitfDevices registered on it. The unit of arbitration is a TRANSACTION: an ordered list of eSteps that a device hands over in one go, executed back to back with the bus held throughout. That is what makes a write and its read-back inseparable - no other device's traffic can land between them - and it is why a meter with three register blocks now wins the bus once per poll round instead of three times. Selection resumes at a cursor rather than restarting at device 0, so the device registered last is served as often as the device registered first. The old loop ran FOR 0 TO count-1 and took the first taker, which is strict priority by registration order dressed up as a scan. Commands are looked for before polls, each pass round-robin from the same cursor, so a Home Assistant command does not queue behind every meter while a chatty device still cannot starve a quiet one. The protocol lives behind I_RS485_TRANSPORT. This block never sees a CRC, a function code or a serial handle. *)
FUNCTION_BLOCK FB_RS485_BUSCONTROLLER
  VAR_OUTPUT
    BusOcupied : BOOL := TRUE;  (* TRUE until the startup delay has passed, then whenever a transaction is in flight *)
    ActiveDevice : INT := -1;  (* Index of the device holding the bus, -1 when free *)
    Cursor : INT;  (* Where the next selection pass starts. Watching this move is how you see fairness working *)
    Transactions : UDINT;  (* Completed transactions since boot *)
    StepsExecuted : UDINT;  (* eSteps attempted; always >= Transactions *)
    StepFailures : UDINT;  (* Of those, how many failed *)
    Watchdogs : UDINT;  (* eSteps abandoned because the transport never answered. Should stay 0 *)
  END_VAR
  VAR
    Transport : I_RS485_TRANSPORT;
    bInitialised : BOOL;
    aitfDevices : ARRAY[0..31] OF I_RS485_DEVICE;
    iDevicesCount : INT;
    StartupDelay : TIME := TIME#5s0ms;  (* Let the slaves finish booting before talking to them *)
    SilenceTime : TIME := TIME#50ms;  (* Quiet between frames, inside a transaction and between them *)
    StepTimeout : TIME := TIME#3s0ms;  (* A step the transport never finishes is abandoned *)
    fbStartupTimer : TON;
    fbSilence : TON;
    fbWatchdog : TON;
    bSilenceRun : BOOL;
    bRestartSilence : BOOL;
    bRestartWatchdog : BOOL;
    iState : INT;  (* 0 idle, 1 execute, 2 collect, 3 gap, 4 release, 5 settle *)
    eSteps : A_RS485_STEP_LIST;
    iStepCount : INT;
    StepIndex : INT;
    StepsRun : INT;
    Failures : INT;
    iChosen : INT;
    eStepState : E_RS485_STEP_STATE;
  END_VAR

            (* Nothing works until Init has supplied a transport. Failing quietly here is
   better than dereferencing a null interface on a running controller. *)
IF NOT bInitialised THEN
	RETURN;
END_IF

(* The transport is serviced every cycle, not only while a step is in flight -
   it is what opens and re-opens the serial port, and it needs cycles to do that
   before anyone asks it to carry anything. *)
eStepState := Transport.Service();

fbStartupTimer(IN := TRUE, PT := StartupDelay);
fbSilence(IN := bSilenceRun AND NOT bRestartSilence, PT := SilenceTime);
fbWatchdog(IN := (iState = 1 OR iState = 2) AND NOT bRestartWatchdog, PT := StepTimeout);
bRestartSilence	:= FALSE;
bRestartWatchdog	:= FALSE;

CASE iState OF

0:	(* ---------------------------------------------------------------- idle *)
	BusOcupied := NOT fbStartupTimer.Q;

	IF fbStartupTimer.Q AND iDevicesCount > 0 THEN
		iChosen := THIS^.SelectNext();
		IF iChosen >= 0 THEN
			ActiveDevice	:= iChosen;
			Cursor			:= (iChosen + 1) MOD iDevicesCount;
			BusOcupied		:= TRUE;

			(* One call, all of this device's work. *)
			iStepCount := aitfDevices[iChosen].BuildTransaction(pSteps := ADR(eSteps));
			IF iStepCount < 0 THEN
				iStepCount := 0;
			ELSIF iStepCount > (DINT_TO_INT(UPPER_BOUND(eSteps, 1)) + 1) THEN
				iStepCount := DINT_TO_INT(UPPER_BOUND(eSteps, 1)) + 1;
			END_IF

			StepIndex	:= 0;
			StepsRun	:= 0;
			Failures	:= 0;

			IF iStepCount = 0 THEN
				(* Withdrew after asking. Release rather than hold the bus. *)
				iState := 4;
			ELSE
				bRestartWatchdog := TRUE;
				iState := 1;
			END_IF
		END_IF
	END_IF

1:	(* ------------------------------------------------- hand the step over *)
	BusOcupied := TRUE;
	IF Transport.Start(pStep := ADR(eSteps[StepIndex])) THEN
		iState := 2;
	ELSIF fbWatchdog.Q THEN
		(* Refused for as long as the fbWatchdog allows: the port is down, or the
		   function code is one this transport will not frame. Either way the
		   step is over - retrying forever would wedge the whole bus. *)
		Watchdogs := Watchdogs + 1;
		THIS^.FinishStep(Failed := TRUE, pData := 0, Count := 0);
	END_IF

2:	(* ------------------------------------------------------ wait it out *)
	BusOcupied := TRUE;
	IF eStepState = E_RS485_STEP_STATE.OK THEN
		THIS^.FinishStep(Failed := FALSE,
		                 pData := Transport.ReadBuffer(),
		                 Count := Transport.Registers());
	ELSIF eStepState = E_RS485_STEP_STATE.FAILED THEN
		THIS^.FinishStep(Failed := TRUE, pData := Transport.ReadBuffer(), Count := 0);
	ELSIF fbWatchdog.Q THEN
		Watchdogs := Watchdogs + 1;
		THIS^.FinishStep(Failed := TRUE, pData := 0, Count := 0);
	END_IF

3:	(* ------------------------ fbSilence between two eSteps of one transaction *)
	(* The bus is NOT released here. This gap is the inter-frame fbSilence RTU
	   needs; letting another device in would break the guarantee that makes a
	   read-after-write worth doing. *)
	BusOcupied := TRUE;
	IF fbSilence.Q THEN
		bSilenceRun		:= FALSE;
		bRestartWatchdog	:= TRUE;
		iState			:= 1;
	END_IF

4:	(* ------------------------------------------------------------- release *)
	BusOcupied := TRUE;
	aitfDevices[ActiveDevice].OnTransactionDone(StepsRun := StepsRun, Failures := Failures);
	Transactions	:= Transactions + 1;
	ActiveDevice	:= -1;
	bSilenceRun		:= TRUE;
	bRestartSilence	:= TRUE;
	iState			:= 5;

5:	(* --------------------------------- fbSilence before anyone else may start *)
	BusOcupied := TRUE;
	IF fbSilence.Q THEN
		bSilenceRun	:= FALSE;
		iState		:= 0;
	END_IF

END_CASE

          

METHOD FinishStep
  VAR_INPUT
    Failed : BOOL;
    pData : POINTER TO A_RS485_READ_BUFFER;
    Count : INT;
  END_VAR
                  (* One step is over, for whatever reason. Report it, then decide whether the
   transaction continues. *)

aitfDevices[ActiveDevice].OnStepResult(StepIndex := StepIndex,
                                   Failed := Failed,
                                   pData := pData,
                                   Count := Count);

StepsRun		:= StepsRun + 1;
StepsExecuted	:= StepsExecuted + 1;

IF Failed THEN
	Failures		:= Failures + 1;
	StepFailures	:= StepFailures + 1;
END_IF

IF Failed AND eSteps[StepIndex].AbortOnError THEN
	(* The step that everything after it depended on. Skipping the rest is the
	   point: a read-back published after a failed write would report a value
	   the device never took. *)
	iState := 4;

ELSE
	StepIndex := StepIndex + 1;
	IF StepIndex >= iStepCount THEN
		iState := 4;
	ELSE
		bSilenceRun		:= TRUE;
		bRestartSilence	:= TRUE;
		iState			:= 3;
	END_IF
END_IF

                
END_METHOD

METHOD SelectNext : INT
  VAR
    iK : INT;
    iI : INT;
  END_VAR
                  (* Round-robin from the cursor, twice: once for work somebody is waiting on,
   once for routine polling.

   Starting each pass at Cursor rather than at 0 is the whole fairness story.
   The loop this replaces ran FOR 0 TO iDevicesCount - 1 and EXITed on the first
   taker, so device 0 won every contested cycle and the device registered last
   only ever got the bus when everything above it was idle. With two meters on
   five-second polls that is invisible; with thirty nodes it is starvation.

   Both passes sweep every device, so a COMMAND anywhere beats a POLL
   everywhere - but COMMANDs are themselves served round-robin, so a chatty
   device cannot monopolise the bus either. *)

SelectNext := -1;

FOR iK := 0 TO iDevicesCount - 1 DO
	iI := (Cursor + iK) MOD iDevicesCount;
	IF aitfDevices[iI].HasWork() = E_RS485_WORK_LEVEL.COMMAND THEN
		SelectNext := iI;
		RETURN;
	END_IF
END_FOR

FOR iK := 0 TO iDevicesCount - 1 DO
	iI := (Cursor + iK) MOD iDevicesCount;
	IF aitfDevices[iI].HasWork() = E_RS485_WORK_LEVEL.POLL THEN
		SelectNext := iI;
		RETURN;
	END_IF
END_FOR

                
END_METHOD

METHOD RegisterDevice : BOOL
  VAR_INPUT
    device : I_RS485_DEVICE;
  END_VAR
                  (* Registration order no longer decides who is served first - that is the point
   of the cursor - so aitfDevices can be registered in whatever order reads best at
   the call site. *)
IF iDevicesCount <= DINT_TO_INT(UPPER_BOUND(aitfDevices, 1)) THEN
	aitfDevices[iDevicesCount]	:= device;
	iDevicesCount			:= iDevicesCount + 1;
	RegisterDevice			:= TRUE;
ELSE
	RegisterDevice := FALSE;
END_IF

                
END_METHOD

METHOD Init
  VAR_INPUT
    Transport : I_RS485_TRANSPORT;  (* The protocol implementation to drive. Replaces the BusTrigger / BusData / BusError pointer trio, which existed only because the framing lived in a program action rather than in a block of its own. *)
    StartupDelay : TIME;  (* Wait this long after a cold start before talking to anything, so slaves that boot slower than the PLC are not written off as missing. Zero keeps the default of 5 s. *)
    SilenceTime : TIME;  (* Quiet line between frames - both between the eSteps of one transaction and between transactions. Zero keeps the default of 50 ms. *)
    StepTimeout : TIME;  (* How long one step may take before the scheduler stops waiting for the transport and moves on. This is a fbWatchdog on the transport, not on the slave; the slave's own reply timeout is shorter and lives in the transport. Zero keeps the default of 3 s. *)
  END_VAR
                  (* Without this, bInitialised went TRUE for a null transport too, and the
   guard on it only ever caught "Init was never called" - not "Init was
   called with nothing to drive", which is the same crash one cycle later. *)
IF Transport = 0 THEN
	RETURN;
END_IF

THIS^.Transport := Transport;

(* Zero means "keep the default", so a call site can supply only what it cares
   about and the block still starts with sane timings. *)
IF StartupDelay > T#0S THEN
	THIS^.StartupDelay := StartupDelay;
END_IF
IF SilenceTime > T#0S THEN
	THIS^.SilenceTime := SilenceTime;
END_IF
IF StepTimeout > T#0S THEN
	THIS^.StepTimeout := StepTimeout;
END_IF

bInitialised := TRUE;

                
END_METHOD

(* How many aitfDevices are registered on this bus. Exists so commissioning can walk the same list the scheduler serves, rather than being handed a second list to keep in step with this one. *)
METHOD DeviceCount : INT
                  DeviceCount := iDevicesCount;

                
END_METHOD

(* The registered device at Index, counted from zero. Read-only access to the list, for anything that has to ask every device on the bus a question - commissioning is the one that does. Index outside the registered range returns nothing rather than whatever is left in the array. *)
METHOD GetDevice : I_RS485_DEVICE
  VAR_INPUT
    Index : INT;
  END_VAR
                  IF Index >= 0 AND Index < iDevicesCount THEN
	GetDevice := aitfDevices[Index];
END_IF

                
END_METHOD
END_FUNCTION_BLOCK

FUNCTION_BLOCK FB_RS485_COMMISSIONER
  VAR_OUTPUT
    Done : BOOL;  (* TRUE once there is nothing left to commission and the bus is back on its own settings. The scheduler must not run until this is TRUE, and it is TRUE on the first cycle when no device asked for anything. *)
    Asked : INT;  (* devices asked whether they need commissioning *)
    Requested : INT;  (* how many said yes *)
    Written : INT;  (* how many were actually changed *)
    Probes : UDINT;  (* Modbus exchanges spent hunting, across all devices *)
    LastReport : STRING(255);
  END_VAR
  VAR
    Transport : I_RS485_TRANSPORT;
    pController : POINTER TO FB_RS485_BUSCONTROLLER;
    BusBaudrate : UDINT;
    pQueue : POINTER TO FB_MQTT_PUBLISH_QUEUE;
    psTopicPrefix : POINTER TO STRING;
    Enabled : BOOL;
    bInitialised : BOOL;
    iState : INT := 0;
    iDeviceIdx : INT := 0;
    device : I_RS485_DEVICE;
    stRequest : ST_RS485_COMMISSION_REQUEST;
    stStep : ST_RS485_STEP;
    fbDelay : TON;
    eOutcome : E_RS485_STEP_STATE;
    iBaudIdx : INT;  (* Per device, reset each time one asks for commissioning. *)
    iStopIdx : INT;
    udiFoundBaud : UDINT;
    byFoundStop : BYTE;
    udiMaxRx : UDINT;
    udiMaxRxBaud : UDINT;
    byMaxRxStop : BYTE;
    udiDeviceProbes : UDINT;
    bDeviceWritten : BOOL;
    sReport : STRING(255);
  END_VAR

            (* Nothing configured, nothing to hold the bus off for. A commissioner that was
   never Init'ed must not stop a bus from working - the failure mode of the
   alternative is a silent bus with no error to show for it. *)
IF NOT bInitialised THEN
	Done := TRUE;
	RETURN;
END_IF

CASE iState OF

0:	IF NOT Enabled OR pController = 0 THEN
		iState := 90;
	ELSE
		iDeviceIdx := 0;
		iState := 1;
	END_IF

1:	(* Ask the next registered device. This is the whole of what makes the sequence
	   device-agnostic: what to probe, what to write and which rates are worth
	   trying all come back from the device itself. *)
	IF iDeviceIdx >= pController^.DeviceCount() THEN
		iState := 90;
	ELSE
		device := pController^.GetDevice(Index := iDeviceIdx);
		Asked := Asked + 1;
		IF device.GetCommissioning(BusBaudrate := BusBaudrate, pRequest := ADR(stRequest)) THEN
			Requested		:= Requested + 1;
			iBaudIdx			:= 0;
			iStopIdx			:= 0;
			udiFoundBaud		:= 0;
			byFoundStop		:= 0;
			udiMaxRx			:= 0;
			udiMaxRxBaud		:= 0;
			byMaxRxStop		:= 0;
			udiDeviceProbes	:= 0;
			bDeviceWritten	:= FALSE;
			iState			:= 2;
		ELSE
			iState := 80;
		END_IF
	END_IF

2:	(* Bring the bus to the setting under test. Short timeouts: a probe that is
	   going to fail should fail quickly, because most of them will. *)
	IF Transport.Retune(
			Baudrate		:= stRequest.Bauds[iBaudIdx],
			StopBitsRaw		:= stRequest.StopBits[iStopIdx],
			ReplyTimeout	:= T#200MS,
			GapTime			:= T#20MS) THEN
		fbDelay(IN := FALSE);
		iState := 3;
	ELSE
		(* A transport that cannot be re-tuned cannot be swept. Give up rather than
		   probe at a setting only believed to be applied. *)
		iState := 70;
	END_IF

3:	(* Let Service actually re-open the port before anything is sent into it. *)
	fbDelay(IN := TRUE, PT := T#200MS);
	Transport.Service();
	IF fbDelay.Q THEN
		fbDelay(IN := FALSE);
		iState := 4;
	END_IF

4:	(* Probe. The point is not what comes back - it is that something did. *)
	stStep.DeviceId		:= stRequest.DeviceId;
	stStep.FunctionCode	:= stRequest.ProbeFunction;
	stStep.Address		:= stRequest.ProbeAddress;
	stStep.Quantity		:= stRequest.ProbeQuantity;
	stStep.AbortOnError	:= FALSE;

	fbDelay(IN := TRUE, PT := T#2S);
	IF Transport.Start(pStep := ADR(stStep)) THEN
		fbDelay(IN := FALSE);
		udiDeviceProbes	:= udiDeviceProbes + 1;
		Probes			:= Probes + 1;
		iState			:= 5;
	ELSIF fbDelay.Q THEN
		(* Port never opened at this setting. A miss, not a fault. *)
		fbDelay(IN := FALSE);
		iState := 6;
	END_IF

5:	eOutcome := Transport.Service();
	IF eOutcome <> E_RS485_STEP_STATE.BUSY THEN
		(* Bytes arriving at all is the useful signal when none of them frame: it
		   separates a device that is present and mis-configured from a bus with
		   nothing on it, which is the difference between sweeping on and going to
		   look at the wiring. *)
		IF Transport.LastRxCount() > udiMaxRx THEN
			udiMaxRx		:= Transport.LastRxCount();
			udiMaxRxBaud	:= stRequest.Bauds[iBaudIdx];
			byMaxRxStop	:= stRequest.StopBits[iStopIdx];
		END_IF
		IF eOutcome = E_RS485_STEP_STATE.OK THEN
			udiFoundBaud	:= stRequest.Bauds[iBaudIdx];
			byFoundStop	:= stRequest.StopBits[iStopIdx];
			iState		:= 7;
		ELSE
			iState := 6;
		END_IF
	END_IF

6:	(* Next rate; when the rates run out, the next framing; when both run out, this
	   device cannot be reached at any setting it named. *)
	IF iBaudIdx < stRequest.BaudCount - 1 THEN
		iBaudIdx	:= iBaudIdx + 1;
		iState	:= 2;
	ELSIF iStopIdx < stRequest.StopCount - 1 THEN
		iBaudIdx		:= 0;
		iStopIdx		:= iStopIdx + 1;
		iState		:= 2;
	ELSE
		iState := 70;
	END_IF

7:	(* Found it. Already where it belongs? Then there is nothing to write, which is
	   the normal eOutcome on every boot after the first. *)
	IF udiFoundBaud = BusBaudrate THEN
		iState := 70;
	ELSE
		iState := 8;
	END_IF

8:	(* Write the value the device asked for into the register it named. Nothing here
	   knows what that value means. *)
	stStep.DeviceId		:= stRequest.DeviceId;
	stStep.FunctionCode	:= stRequest.WriteFunction;
	stStep.Address		:= stRequest.WriteAddress;
	stStep.Quantity		:= 1;
	stStep.Data[0]		:= stRequest.WriteValue;
	stStep.AbortOnError	:= FALSE;

	fbDelay(IN := TRUE, PT := T#2S);
	IF Transport.Start(pStep := ADR(stStep)) THEN
		fbDelay(IN := FALSE);
		bDeviceWritten	:= TRUE;
		Written			:= Written + 1;
		iState			:= 9;
	ELSIF fbDelay.Q THEN
		fbDelay(IN := FALSE);
		iState := 70;
	END_IF

9:	(* The acknowledgement comes back at the NEW setting and this end will not hear
	   it, so the eOutcome is deliberately ignored: a failure here is the expected
	   result of success, and nothing may retry on it. *)
	IF Transport.Service() <> E_RS485_STEP_STATE.BUSY THEN
		iState := 70;
	END_IF

70:	(* Put the bus back the way the program configured it, whatever happened. *)
	Transport.RestoreTuning();
	fbDelay(IN := FALSE);
	iState := 71;

71:	fbDelay(IN := TRUE, PT := T#500MS);
	Transport.Service();
	IF fbDelay.Q THEN
		fbDelay(IN := FALSE);
		iState := 72;
	END_IF

72:	(* Publish the eOutcome, retained, so it can be read off the broker at any time.
	   The alternative is an online debug session, and on this hardware that is the
	   least reliable thing in the chain - the runtime drops the session long before
	   it drops MQTT. A commissioning result nobody can read is not a result.

	   Built up a piece at a time rather than nested: CONCAT takes exactly two
	   arguments, and a seven-deep nest of it is unreadable even when correct. *)
	sReport := CONCAT('probes=', UDINT_TO_STRING(udiDeviceProbes));
	sReport := CONCAT(sReport, ' found=');
	sReport := CONCAT(sReport, UDINT_TO_STRING(udiFoundBaud));
	sReport := CONCAT(sReport, '/');
	sReport := CONCAT(sReport, BYTE_TO_STRING(byFoundStop));
	sReport := CONCAT(sReport, ' maxrx=');
	sReport := CONCAT(sReport, UDINT_TO_STRING(udiMaxRx));
	sReport := CONCAT(sReport, ' at=');
	sReport := CONCAT(sReport, UDINT_TO_STRING(udiMaxRxBaud));
	sReport := CONCAT(sReport, '/');
	sReport := CONCAT(sReport, BYTE_TO_STRING(byMaxRxStop));
	sReport := CONCAT(sReport, ' written=');
	sReport := CONCAT(sReport, BOOL_TO_STRING(bDeviceWritten));
	LastReport := sReport;

	IF pQueue <> 0 AND psTopicPrefix <> 0 AND stRequest.ReportTopic <> '' THEN
		pQueue^.AddMessageOn(Lane := GVL_MQTT.MQTT_LANE_RS485,
			Payload := sReport,
			Topic := CONCAT(psTopicPrefix^, stRequest.ReportTopic),
			Qos := MQTT.QoS.ExactlyOnce,
			MqttRetain := TRUE);
	END_IF

	iState := 80;

80:	iDeviceIdx	:= iDeviceIdx + 1;
	iState		:= 1;

90:	(* Nothing left to do. The bus is on its own settings and the scheduler can
	   have it. *)
	Done := TRUE;

END_CASE

          

(* Wires the commissioner to the bus it is to look after. Call once at startup, after every device has been registered with the bus controller - the list is read through the controller so there is only ever one of it. *)
METHOD Init
  VAR_INPUT
    Transport : I_RS485_TRANSPORT;  (* The bus. Re-tuned during a sweep and restored afterwards, which is why it is the transport interface rather than a port number. *)
    pController : POINTER TO FB_RS485_BUSCONTROLLER;  (* Bus controller holding the registered devices. Commissioning asks the same list the scheduler serves, so nothing can be commissioned that is not polled, or polled that was not commissioned. *)
    BusBaudrate : UDINT;  (* What this bus runs at. Passed to each device so it can encode that rate the way its own register expects, and so a device already at it is left alone. *)
    pMqttPublishQueue : POINTER TO FB_MQTT_PUBLISH_QUEUE;  (* Queue the retained result is published on. Zero publishes nothing and commissions all the same. *)
    MqttPublishPrefix : POINTER TO STRING;  (* Topic prefix the device's own ReportTopic is appended to. *)
    Enable : BOOL;  (* FALSE skips commissioning entirely and releases the bus on the first cycle. *)
  END_VAR
                  THIS^.Transport		:= Transport;
THIS^.pController	:= pController;
THIS^.BusBaudrate	:= BusBaudrate;
THIS^.pQueue		:= pMqttPublishQueue;
THIS^.psTopicPrefix	:= MqttPublishPrefix;
THIS^.Enabled		:= Enable;

bInitialised := TRUE;

                
END_METHOD
END_FUNCTION_BLOCK

{attribute 'reflection'}
FUNCTION_BLOCK FB_RS485_DFROBOT_SEN0492_MQTT EXTENDS FB_MQTT_BASE IMPLEMENTS I_RS485_DEVICE
  VAR CONSTANT
    ctSen0492MinPoll : TIME := TIME#8s0ms;  (* Measured floor for this sensor, not a guess: it answers about once every six to seven seconds however often it is asked, so anything faster only raises the proportion of requests that fail. See FB_init. *)
  END_VAR
  VAR
    {attribute 'noinit'}
    {attribute 'instance-path'}
    sInstancePath : STRING(GVL_MQTT.MQTT_TOPIC_LEN);  (* object's full instance name *)
    stStep : ST_RS485_STEP;  (* The one register block this sensor is read in: distance and output state are adjacent, so one request gets both and they are guaranteed to describe the same measurement. Filled by FB_init in iCode rather than by a declaration initialiser - a value inside an existing structured initialiser cannot be changed from a script afterwards. *)
    stConfigStep : ST_RS485_STEP;  (* A pending configuration write. The sensor's settings live in ordinary holding registers, so changing one is an FC6 stStep like any other - it just has to jump the polling queue, which is what E_RS485_WORK_LEVEL.COMMAND is for. See RequestConfigWrite. *)
    bConfigPending : BOOL := FALSE;
    fbTimerData : TON;
    bIsDataUpdated : BOOL := FALSE;
    bIsStateUpdated : BOOL := FALSE;
    iAvailFailures : INT := 0;  (* Availability is a judgement, not a reading. One missed reply on a shared RS485 bus is ordinary - a slave that was mid-measurement, a collision with another device's turnaround - and publishing 'offline' on the strength of it makes the Home Assistant connectivity sensor flap between states that are both wrong. So failures have to accumulate before the device is declared down, and recovery is immediate on the first good transaction: being slow to trust and quick to forgive is the right asymmetry when the cost of a false 'offline' is an entity that looks broken. *)
    bAvailOnline : BOOL := FALSE;
    bAvailKnown : BOOL := FALSE;
    abQualityWindow : ARRAY[0..15] OF BOOL;  (* Quality, which is a different question from availability and needs a different answer. Availability is binary and has to be debounced or it reports noise; that same debounce means a sensor answering two polls in three still reads 'online', which is true and useless. This is the signal that says how well it is working rather than whether it is: the share of the last sixteen transactions that succeeded, as a percentage. A sensor degrading - a loose pair, a failing driver, a bus getting busier - shows up here long before it shows up as a disconnection. *)
    iQualityIdx : INT := 0;
    iQualitySeen : INT := 0;
    bIsQualityUpdated : BOOL := FALSE;
    fbMqttDiscoveryDevice : FB_DFROBOT_MQTT_DISCOVERY_DEVICE;  (* The sensor announced to Home Assistant as a device of its own. One per sensor and its lifetime is the sensor's, so it lives here rather than in a GVL - the Eastron meters do the same. *)
  END_VAR
  VAR_INPUT
    PollIntervalOverride : TIME := TIME#0ms;  (* The poll interval that can actually be changed without the IDE. FB_init's DataPollingInterval is the default and it is the honest place for it, but CODESYS stores an instance's FB_init arguments outside the declaration text, so no script can revise one - see CLAUDE.md. That makes the constructor argument a one-way door for tooling, which is awkward for the one number on this block most likely to need tuning. So: zero means use whatever FB_init was given; anything else wins, subject to the same ctSen0492MinPoll floor. Settable from RS485_INIT, or online while the PLC runs. *)
    AvailabilityFailLimit : INT := 3;  (* Consecutive failed transactions before this device is declared offline. Three is about six seconds at the default two-second poll. Raise it on a bus that is busy or long; one would mean every transient shows up in Home Assistant as a disconnection. *)
  END_VAR
  VAR_OUTPUT
    DISTANCE : UINT := 0;  (* Millimetres, straight from the sensor - it reports an integer and there is no scaling to undo. Only updated while OUTPUT_STATE says the reading is good, so a failed measurement holds the last trustworthy distance rather than replacing it with a plausible-looking wrong one. *)
    OUTPUT_STATE : BYTE := 0;  (* 0 = valid; 1 sigma fail, 2 signal fail, 3 min range fail, 4 phase fail, 5 hardware fail, 7 no update. Published on every poll whatever it says, because it is the only thing that explains a distance that stopped moving. *)
    MeasurementValid : BOOL := FALSE;
    DataAvailable : BOOL := FALSE;
    Error : BOOL := FALSE;
    SuccessRate : USINT := 100;  (* Percentage of the last sixteen transactions that succeeded. 100 is a healthy sensor; anything settling below that is worth looking at even while availability still reads online. *)
  END_VAR

            (* --- self-wiring prologue ----------------------------------------------------
   Makes the InitMqtt and InitMqttDiscovery calls optional. Set FriendlyName at
   the declaration site and this block wires itself from GVL_MQTT on its
   first cyclic call, then announces itself to Home Assistant.

   Deliberately in the body rather than in FB_init: it dereferences GVL members
   and reads the reflection instance path, and doing that during initialisation
   would rely on an ordering nothing enforces and the compiler cannot check.

   Dormant while FriendlyName is empty, so a call site that wires the block by
   hand keeps working untouched. A block wired this way MUST be called
   cyclically, and nothing warns if it is not. *)
IF FriendlyName <> '' THEN

	IF NOT bInitMqttDone THEN
		THIS^.InitMqtt(
			MQTTPublishPrefix := ADR(GVL_MQTT.MqttPubRS485Prefix),
			pMqttPublishQueue := ADR(GVL_MQTT.fbMqttPublishQueue));
	END_IF

	IF bInitMqttDone AND NOT bInitMqttDiscoveryDone THEN
		THIS^.InitMqttDiscovery(
			Device := ADR(THIS^.fbMqttDiscoveryDevice),
			DeviceName := FriendlyName);
	END_IF

END_IF

(* Applied every cycle rather than once, so the interval can be changed online
   and take effect on the next poll. Below the floor is raised to it, exactly as
   FB_init does - a limit worth enforcing is worth enforcing on both routes in. *)
IF PollIntervalOverride > T#0S THEN
	IF PollIntervalOverride < ctSen0492MinPoll THEN
		fbTimerData.PT := ctSen0492MinPoll;
	ELSE
		fbTimerData.PT := PollIntervalOverride;
	END_IF
END_IF

fbTimerData();

(* The state goes out on every poll and the distance only when the sensor called
   it valid, so a reader can always tell a held reading from a fresh one. *)
IF bIsStateUpdated THEN
	bIsStateUpdated := FALSE;
	PubMqttMessage(Suffix := '/STATE', Data := BYTE_TO_STRING(OUTPUT_STATE));
END_IF

IF bIsDataUpdated THEN
	bIsDataUpdated := FALSE;
	PubMqttMessage(Suffix := '/DIST', Data := UINT_TO_STRING(DISTANCE));
END_IF

(* Published on every transaction, unlike availability: a slowly falling number
   is exactly the signal this exists to carry, and suppressing the unchanged
   values would hide a sensor sitting steadily at 60%. *)
IF bIsQualityUpdated THEN
	bIsQualityUpdated := FALSE;
	PubMqttMessage(Suffix := '/QUALITY', Data := USINT_TO_STRING(SuccessRate));
END_IF

          

METHOD RequestConfigWrite : BOOL
  VAR_INPUT
    Register : UINT;  (* Holding register to write. 16#04 baud rate, 16#1A slave id, 16#08 measurement interval, 16#36 measurement mode, 16#00 factory reset. *)
    Value : WORD;  (* Value to write. For the baud rate register, 0..9 selects 2400 through 921600; 2 is 9600. *)
  END_VAR
                  (* Queues a single-register write for the next time this device is granted the
   bus. HasWork reports COMMAND while one is pending, so it goes ahead of routine
   polling on this and every other device.

   Registers worth knowing, from the DFRobot reference:
     16#04  baud rate    0..9 = 2400, 4800, 9600, 19200, 38400, 57600,
                         115200, 230400, 460800, 921600
     16#1A  slave id     16#00..16#FE
     16#08  measurement interval, 1..1000 ms
     16#36  measurement mode  1 = up to 1.3 m, 2 = up to 3 m, 3 = up to 4 m
     16#00  write 1 to restore factory settings

   Writing the baud rate takes effect immediately, so the sensor answers - if at
   all - at the NEW rate and this end will not hear it. That is expected and is
   why OnTransactionDone does not retry. *)
IF NOT bConfigPending THEN
	stConfigStep.DeviceId		:= stStep.DeviceId;
	stConfigStep.FunctionCode	:= 6;
	stConfigStep.Address		:= Register;
	stConfigStep.Quantity		:= 1;
	stConfigStep.Data[0]		:= Value;
	stConfigStep.AbortOnError	:= FALSE;
	bConfigPending			:= TRUE;
	RequestConfigWrite		:= TRUE;
ELSE
	RequestConfigWrite		:= FALSE;
END_IF

                
END_METHOD

METHOD OnTransactionDone
  VAR_INPUT
    StepsRun : INT;
    Failures : INT;
  END_VAR
  VAR
    iQualityOk : INT;
    iQualityI : INT;
  END_VAR
                  (* One decision per transaction, and one re-arm of the timer.

   The re-arm belongs here rather than in OnStepResult because a stStep skipped by
   an AbortOnError predecessor is never reported, and a sensor that has stopped
   answering must still be retried. OnTransactionDone always runs. *)
fbTimerData.IN := TRUE;

(* A configuration write is finished either way. It is deliberately not retried:
   the write that changes the baud rate cannot be confirmed at the old baud rate,
   so a retry loop here would spin forever on a sensor that had in fact obeyed.
   It also says nothing about availability - a write that cannot be acknowledged
   is not evidence the sensor has gone away. *)
IF bConfigPending THEN
	bConfigPending := FALSE;
	RETURN;
END_IF

IF StepsRun = 0 THEN
	RETURN;
END_IF

(* Two independent verdicts on the same transaction, because they answer
   different questions. iAvailFailures decides whether the sensor is reachable at
   all and needs hysteresis to be worth reading. The quality window records how
   well it is doing and deliberately has none - the whole point is to move while
   availability is still, so that a sensor which is degrading rather than
   disconnected is visible. *)
IF Failures >= StepsRun THEN
	IF iAvailFailures < AvailabilityFailLimit THEN
		iAvailFailures := iAvailFailures + 1;
	END_IF
	abQualityWindow[iQualityIdx] := FALSE;
ELSE
	iAvailFailures := 0;
	abQualityWindow[iQualityIdx] := TRUE;
END_IF

iQualityIdx := (iQualityIdx + 1) MOD (DINT_TO_INT(UPPER_BOUND(abQualityWindow, 1)) + 1);
IF iQualitySeen <= DINT_TO_INT(UPPER_BOUND(abQualityWindow, 1)) THEN
	iQualitySeen := iQualitySeen + 1;
END_IF

(* Only over what has actually been observed, so the figure is honest from the
   first transaction rather than starting at a flattering 100 for sixteen. *)
iQualityOk := 0;
FOR iQualityI := 0 TO iQualitySeen - 1 DO
	IF abQualityWindow[iQualityI] THEN
		iQualityOk := iQualityOk + 1;
	END_IF
END_FOR

IF iQualitySeen > 0 THEN
	SuccessRate := INT_TO_USINT((iQualityOk * 100) / iQualitySeen);
	bIsQualityUpdated := TRUE;
END_IF

(* Published only when the verdict changes, and once at startup so a retained
   value exists before anything has gone wrong. Republishing 'online' every two
   seconds for the life of the PLC tells nobody anything and is most of the
   traffic this block would otherwise generate. *)
IF iAvailFailures >= AvailabilityFailLimit THEN
	IF bAvailOnline OR NOT bAvailKnown THEN
		bAvailOnline := FALSE;
		bAvailKnown := TRUE;
		PubMqttMessage(Suffix := '/availability', Data := 'offline');
	END_IF
ELSIF iAvailFailures = 0 THEN
	IF NOT bAvailOnline OR NOT bAvailKnown THEN
		bAvailOnline := TRUE;
		bAvailKnown := TRUE;
		PubMqttMessage(Suffix := '/availability', Data := 'online');
	END_IF
END_IF

                
END_METHOD

METHOD OnStepResult
  VAR_INPUT
    StepIndex : INT;
    Failed : BOOL;
    pData : POINTER TO A_RS485_READ_BUFFER;
    Count : INT;
  END_VAR
                  (* A configuration write echoes the request back rather than returning data; the
   transport has already checked that echo, so there is nothing to decode here. *)
IF bConfigPending THEN
	RETURN;
END_IF

THIS^.Error := Failed;

(* Count is what actually came back, not what was asked for, so a short reply
   cannot be read past the end of. *)
IF NOT Failed AND Count >= 2 THEN
	THIS^.OUTPUT_STATE		:= WORD_TO_BYTE(pData^[1] AND 16#00FF);
	THIS^.MeasurementValid	:= (THIS^.OUTPUT_STATE = 0);
	THIS^.bIsStateUpdated	:= TRUE;

	(* Hold the last good distance rather than publishing one the sensor has
	   just told us not to trust. A stale reading is visibly stale next to a
	   state that is not 'valid'; a wrong one is not visible at all. *)
	IF THIS^.MeasurementValid THEN
		THIS^.DISTANCE		:= WORD_TO_UINT(pData^[0]);
		THIS^.DataAvailable	:= TRUE;
		THIS^.bIsDataUpdated	:= TRUE;
	END_IF
END_IF

                
END_METHOD

METHOD BuildTransaction : INT
  VAR_INPUT
    pSteps : POINTER TO A_RS485_STEP_LIST;
  END_VAR
                  (* A configuration write goes alone and goes first. It is not batched with the
   read because several of these registers change how the sensor talks - the
   baud rate register is the obvious one - and a read queued behind such a write
   would be sent into a sensor that has already stopped listening at this speed. *)
IF bConfigPending THEN
	pSteps^[0]			:= stConfigStep;
	BuildTransaction	:= 1;
ELSIF fbTimerData.Q THEN
	fbTimerData.IN		:= FALSE;
	pSteps^[0]			:= stStep;
	BuildTransaction	:= 1;
ELSE
	BuildTransaction	:= 0;
END_IF

                
END_METHOD

METHOD HasWork : E_RS485_WORK_LEVEL
                  (* Predicate only - the scheduler calls this on every device every cycle, and
   twice when it is looking for commands first. Nothing here may change state. *)
IF bConfigPending THEN
	HasWork := E_RS485_WORK_LEVEL.COMMAND;
ELSIF fbTimerData.Q THEN
	HasWork := E_RS485_WORK_LEVEL.POLL;
ELSE
	HasWork := E_RS485_WORK_LEVEL.NONE;
END_IF

                
END_METHOD

METHOD InitMqttDiscovery
  VAR_INPUT
    Device : POINTER TO FB_DFROBOT_MQTT_DISCOVERY_DEVICE;
    DeviceName : STRING(50);
    Model : STRING(20) := 'SEN0492';
    overruleId : STRING(255) := '';
  END_VAR
  VAR
    id : STRING(255);
  END_VAR
                  (* Announces the sensor as a device of its own, then one entity per thing it
   reports. Distance carries no StateClass: it is a position, not a quantity
   worth averaging or totalling, and Home Assistant's long-term statistics on it
   would be meaningless. *)
IF bInitMqttDone AND NOT bInitMqttDiscoveryDone THEN

	id := SUPER^.ResolveEntityId(overruleId := overruleId);

	Device^.initDFRobotDevice(
		name := DeviceName,
		id := id,
		Model := Model,
		availabilityTopic1 := GVL_MQTT.MqttAvailabilityTopic,
		availabilityTopic2 := CONCAT(THIS^.sMQTTPublishTopic, '/availability'),
		availabilityOnline := GVL_MQTT.MqttAvailabilityOnlinePayload,
		availabilityOffline := GVL_MQTT.MqttAvailabilityOfflinePayload,
		MqttDiscoveryPrefix := GVL_MQTT.MqttHADiscoveryPrefix,
		MqttDiagnosticTopic := CONCAT(THIS^.sMQTTPublishTopic, '/diagnostic'),
		pMqttPublishQueue := ADR(GVL_MQTT.fbMqttPublishQueue));

(* This device publishes from the RS485 task, so its messages take that
   task's queue lane. A lane may only ever have one producing task. *)
Device^.SetLane(Lane := GVL_MQTT.MQTT_LANE_RS485);

	Device^.CreateSensorEntity(
		Name := 'Distance',
		Id := CONCAT(id, '_DIST'),
		StateTopic := CONCAT(THIS^.sMQTTPublishTopic, '/DIST'),
		DeviceClass := 'distance',
		UnitOfMeasurement := 'mm');

	(* Diagnostic rather than a headline reading: it is what you look at when the
	   distance stops making sense, not something to put on a dashboard. *)
	Device^.CreateDiagnosticSensorEntity(
		Name := 'Measurement state',
		Id := CONCAT(id, '_STATE'),
		StateTopic := CONCAT(THIS^.sMQTTPublishTopic, '/STATE'));

	(* Diagnostic, with a unit and a state class so Home Assistant will graph it
	   and keep statistics. This is the entity to put an automation on: a sensor
	   that starts answering nine polls in ten instead of ten shows up here
	   while availability is still reporting a cheerful 'online'. *)
	Device^.CreateDiagnosticSensorEntity(
		Name := 'Link quality',
		Id := CONCAT(id, '_QUALITY'),
		StateTopic := CONCAT(THIS^.sMQTTPublishTopic, '/QUALITY'),
		StateClass := 'measurement',
		UnitOfMeasurement := '%');

	bInitMqttDiscoveryDone := TRUE;
END_IF

                
END_METHOD

METHOD PubMqttMessage
  VAR_INPUT
    Suffix : STRING(100);
    Data : STRING(100);
  END_VAR
                  IF bInitMqttDone THEN
		pMqttPublishQueue^.AddMessageOn(Lane := GVL_MQTT.MQTT_LANE_RS485,
			Payload := Data,
			Topic := CONCAT(THIS^.sMQTTPublishTopic, Suffix),
			Qos := MQTT.QoS.ExactlyOnce,
			MqttRetain := FALSE
		);
END_IF

                
END_METHOD

METHOD InitMqtt
  VAR_INPUT
    MQTTPublishPrefix : POINTER TO STRING;
    pMqttPublishQueue : POINTER TO FB_MQTT_PUBLISH_QUEUE;
  END_VAR
                  SUPER^._sInstancePath := THIS^.sInstancePath; // Due to reflection its location is important

(*pass trough*)
THIS^.pMqttPublishQueue := pMqttPublishQueue;
THIS^.psMqttPublishTopicPrefix := MQTTPublishPrefix;
SUPER^.InitBaseMqtt();

                
END_METHOD

METHOD FB_init : BOOL
  VAR_INPUT
    bInitRetains : BOOL;  (* TRUE: the retain variables are initialized (reset warm / reset cold) *)
    bInCopyCode : BOOL;  (* TRUE: the instance will be copied to the copy iCode afterward (online change) *)
    DeviceAddress : BYTE;  (* Modbus slave address of the sensor. Factory default is 16#50. *)
    DataPollingInterval : TIME;  (* How often the sensor is read. One read covers distance and measurement state. *)
  END_VAR
                  (* Modbus address and poll rate describe the wiring, not a mode, so they are
   fixed for the life of the instance and belong here rather than in a runtime
   setter. Note the consequence: changing either afterwards means editing the
   declaration in the IDE - CODESYS stores an instance's FB_init arguments beside
   the declaration text, where no script can reach them.

   16#34 is the measurement data register and 16#35 the output state; they are
   adjacent, so reading two registers gets both from one reply and they describe
   the same measurement rather than two moments a poll apart.

   Function 3, not 4: this sensor exposes everything - readings and settings
   alike - as holding registers. *)
THIS^.stStep.DeviceId		:= DeviceAddress;
THIS^.stStep.FunctionCode	:= 3;
THIS^.stStep.Address		:= 16#34;
THIS^.stStep.Quantity		:= 2;

(* --- the poll rate is a hardware limit, not a preference --------------------
   This sensor will not be read every two seconds. Measured on a PFC200 with the
   sensor alone on the bus, nothing else registered:

     poll every 2 s   ~19 requests per 30 s, ~4 answered   - 25% success
     poll every 7 s   ~4 requests per 30 s, ~4 answered    - 100%
     poll every 10 s  3 requests per 30 s, 3 answered      - 100%, zero failures

   It answers roughly once every six or seven seconds however often it is asked,
   and the requests in between are simply dropped. Ask faster and the only thing
   that changes is the proportion that fail, which is what made the Home
   Assistant connectivity sensor flap: three consecutive misses is easy to reach
   at 2 s and impossible at 10 s.

   So the interval is clamped rather than trusted. A caller asking for something
   this device cannot sustain gets a working sensor and a slower one, which is
   the better failure: the alternative is a reading that is right a quarter of
   the time and an entity that keeps going unavailable. *)
IF DataPollingInterval < ctSen0492MinPoll THEN
	THIS^.fbTimerData.PT := ctSen0492MinPoll;
ELSE
	THIS^.fbTimerData.PT := DataPollingInterval;
END_IF
THIS^.fbTimerData.IN := TRUE;

FB_init := TRUE;

                
END_METHOD

(* This sensor ships at 115200 baud with no switch on it, so on a bus running at any other rate it is not slow to answer - it is inaudible. That is what there is to commission here, and describing it is the sensor's own business: which register holds the rate, what iCode that register wants for the bus rate, and which rates the register can select at all. See I_RS485_DEVICE.GetCommissioning for the contract. *)
METHOD GetCommissioning : BOOL
  VAR_INPUT
    BusBaudrate : UDINT;
    pRequest : POINTER TO ST_RS485_COMMISSION_REQUEST;
  END_VAR
  VAR
    iI : INT;
    iN : INT;
    iCode : INT;
  END_VAR
  VAR CONSTANT
    caudiBaudRates : ARRAY[0..9] OF UDINT := [2400, 4800, 9600, 19200, 38400, 57600, 115200, 230400, 460800, 921600];  (* Register 16#04 takes a iCode, not a rate - and the iCode is the index into this table, which is why the table is the only place either has to be written down. *)
    cudiFactoryBaud : UDINT := 115200;
    cuiRegBaudrate : UINT := 16#4;
  END_VAR
                  IF pRequest = 0 THEN
	GetCommissioning := FALSE;
	RETURN;
END_IF

(* Can this sensor even be told to use the bus rate? The iCode is the index of the
   rate in its own table, so a rate that is not in the table has no iCode, and the
   honest answer is then to withdraw: moving the sensor to a rate it can express
   but the bus does not use would leave it just as inaudible, at a setting nobody
   went looking for. *)
iCode := -1;
FOR iI := 0 TO DINT_TO_INT(UPPER_BOUND(caudiBaudRates, 1)) DO
	IF caudiBaudRates[iI] = BusBaudrate THEN
		iCode := iI;
	END_IF
END_FOR

IF iCode < 0 THEN
	GetCommissioning := FALSE;
	RETURN;
END_IF

(* Where to probe, and what a reply means. Everything on this sensor - readings and
   settings alike - is a holding register, so it is function 3 to read and 6 to
   write. The probe is the same measurement read the block polls with, because the
   point is not the distance: it is that something answered at this setting. *)
pRequest^.DeviceId			:= stStep.DeviceId;
pRequest^.ProbeFunction		:= 3;
pRequest^.ProbeAddress		:= stStep.Address;
pRequest^.ProbeQuantity		:= stStep.Quantity;
pRequest^.WriteFunction		:= 6;
pRequest^.WriteAddress		:= cuiRegBaudrate;
pRequest^.WriteValue		:= INT_TO_WORD(iCode);

(* The bus rate first, so a sensor that has already been moved costs one exchange
   and the sweep ends there - the normal case after the first successful boot. The
   factory rate second, because that is where a fresh or factory-reset sensor is.
   Then the rest, for a sensor somebody has left half-configured. *)
pRequest^.Bauds[0] := BusBaudrate;
iN := 1;
IF cudiFactoryBaud <> BusBaudrate THEN
	pRequest^.Bauds[iN] := cudiFactoryBaud;
	iN := iN + 1;
END_IF
FOR iI := 0 TO DINT_TO_INT(UPPER_BOUND(caudiBaudRates, 1)) DO
	IF caudiBaudRates[iI] <> BusBaudrate AND caudiBaudRates[iI] <> cudiFactoryBaud THEN
		pRequest^.Bauds[iN] := caudiBaudRates[iI];
		iN := iN + 1;
	END_IF
END_FOR
pRequest^.BaudCount := iN;

(* Framing as well as rate, because those are the two things that silence a device
   on a working pair. 255 leaves the port's own framing - the ordinary case, tried
   first - and 1..3 force the raw SysCom iCode, which is how two stop bits is
   reached without depending on an enumerator name this runtime may spell
   differently. The sensor's own forum traffic reports 8N2; this bench found one
   stop bit answering on the first probe, so the sweep keeps both. *)
pRequest^.StopBits[0]	:= 255;
pRequest^.StopBits[1]	:= 1;
pRequest^.StopBits[2]	:= 2;
pRequest^.StopBits[3]	:= 3;
pRequest^.StopCount		:= 4;

(* Where the outcome is published, retained, under the bus prefix. *)
pRequest^.ReportTopic := 'SEN0492_COMMISSION';

GetCommissioning := TRUE;

                
END_METHOD
END_FUNCTION_BLOCK

{attribute 'reflection'}
FUNCTION_BLOCK FB_RS485_DUCO_DUCOBOX_FOCUS_MQTT EXTENDS FB_MQTT_BASE IMPLEMENTS I_RS485_DEVICE, MQTT.MQTT_SUBSCRIBE_CALLBACK
  VAR
    {attribute 'noinit'}
    {attribute 'instance-path'}
    sInstancePath : STRING(GVL_MQTT.MQTT_TOPIC_LEN);  (* object's full instance name *)
    bStartup : BOOL := TRUE;
    bInitRS485Done : BOOL := FALSE;
    fbTimerData : TON;
    bIsDataUpdated : BOOL := FALSE;
    afbNodes : ARRAY[2..30] OF FB_RS485_DUCO_DUCOBOX_FOCUS_NODE_MQTT;
    uiNodePointer : UINT := 2;
    iLoopCounter : INT;  (* the body's node-call loop *)
    iNodeCursor : INT := 2;  (* Where the next node scan resumes. afbNodes take one slot per transaction and take it in turn, so node 30 is polled as often as node 2 - batching all the due ones would hold the bus for thirty frames and starve the meters. *)
    aiStepMap : ARRAY[0..7] OF INT;  (* What each step of the current transaction is for: 1 the master unit, 2 the write, 3 the read-back of that write, 10 + iN a node. The scheduler hands StepIndex back and this is how it is decoded - the old ActiveNode tag could only describe one thing at a time, which is why a write and a read could not be in flight together. *)
    stMasterStep : ST_RS485_STEP;
    stWriteStep : ST_RS485_STEP;
    stReadBackStep : ST_RS485_STEP;
    bWriteQueryReady : BOOL := FALSE;
    sWriteQuerySuffix : STRING;
    sWriteQueryPayload : STRING;
  END_VAR
  VAR_OUTPUT
    ACTIVEPOWER : REAL := 0;
    DataAvailable : BOOL := FALSE;
    Error : BOOL := FALSE;
  END_VAR
  VAR
    fbMqttDiscoveryDevice : FB_BASE_MQTT_DISCOVERY_DEVICE;  (* This block's own Home Assistant device object, re-pointed at each component in turn before its entities are created. One object rather than one per node: the discovery base carries eighteen config structs and twenty-nine copies of those would not fit. *)
    sDeviceId : STRING(255);
    bTxHadRequiredStep : BOOL := FALSE;  (* Availability is published only when it changes, and only judged on a transaction that carried a step which actually matters. A zone read is optional; letting one condemn the device made Home Assistant blink. *)
    bAvailable : BOOL := FALSE;
    bAvailabilityPublished : BOOL := FALSE;
    bLastAvailable : BOOL := FALSE;
    stLocStep : ST_RS485_STEP;
    fbAvailTick : TON;  (* Availability is counted here and decided on a heartbeat, not per transaction. See OnTransactionDone and the body. *)
    uiTxOk : UINT := 0;
    uiTxSeen : UINT := 0;
    iLastStepsRun : INT := -1;  (* Diagnostics for the availability question. Published on the heartbeat, so the arithmetic can be read off the broker instead of inferred. *)
    iLastFailures : INT := -1;
    uiTxCalls : UINT := 0;
    uiAvailPubs : UINT := 0;
    sAvailDiag : STRING(120);
    awLastMaster : ARRAY[0..5] OF WORD;  (* Last raw master frame, so the six unit topics are only republished when one of them actually moves. See OnStepResult. *)
    bMasterPublished : BOOL := FALSE;
    bRefreshDue : BOOL := TRUE;
    iMasterChk : INT;
    bMasterChanged : BOOL;
    fbMasterRefresh : TON;
    sPayload : STRING(80);  (* Command payload, split so a leading minus can be handled explicitly. See PublishReceived. *)
    sDigits : STRING(80);
    bNegative : BOOL;
    wBoxSettingsMask : WORD := 16#61;  (* The box announces a target position and an auto minimum and maximum - registers 0, 5 and 6 - so those are read back the same way a component's are. Register 9 is the action, which has no readable counterpart. *)
    iBoxSettingsCursor : INT := 0;
    iBoxSettingsPending : INT := -1;
    bBoxSettingsDue : BOOL := TRUE;
    stBoxSettingsStep : ST_RS485_STEP;
    iB : INT;
  END_VAR

            (* --- self-wiring prologue ----------------------------------------------------
   Makes the InitMqtt and InitMqttDiscovery calls optional. Set FriendlyName at
   the declaration site and this block wires itself from GVL_MQTT on its first
   cyclic call, then announces itself and, as the bus reports what they are, each
   of its components.

   In the body rather than in FB_init: it dereferences GVL members, and doing
   that during initialisation would rely on an ordering nothing enforces and the
   compiler cannot check.

   The components are unaffected either way - AddNode carries their names, and a
   component is announced when its type resolves, not when the box is wired.

   Dormant while FriendlyName is empty, so a call site that makes both calls
   itself keeps working untouched.

   A block wired this way MUST be called cyclically. An instance whose body never
   runs is unwired and absent from Home Assistant, and nothing warns about it. *)
IF FriendlyName <> '' THEN

	IF NOT bInitMqttDone THEN
		THIS^.InitMqtt(
			MQTTPublishPrefix := ADR(GVL_MQTT.MqttPubRS485Prefix),
			MQTTSubscribePrefix := ADR(GVL_MQTT.MqttSubRS485Prefix),
			pMqttPublishQueue := ADR(GVL_MQTT.fbMqttPublishQueue),
			pMqttCallbackCollector := ADR(GVL_MQTT.collector_FB_RS485_MQTT));
	END_IF

	IF bInitMqttDone AND NOT bInitMqttDiscoveryDone THEN
		THIS^.InitMqttDiscovery(DeviceName := FriendlyName, overruleId := '');
	END_IF
END_IF

fbTimerData();

FOR iLoopCounter := 2 TO 30 DO
	afbNodes[iLoopCounter]();
END_FOR

(* At most one component announced per cycle. A component's entity set runs to
   about twenty configs, so announcing a whole system at once would put several
   hundred messages into the publish queue in a single cycle. *)
IF bInitMqttDiscoveryDone THEN
	FOR iLoopCounter := 2 TO 30 DO
		IF iLoopCounter < UINT_TO_INT(uiNodePointer) THEN
			IF afbNodes[iLoopCounter].NeedsAnnounce() THEN
				THIS^.AnnounceNode(iN := iLoopCounter);
				EXIT;
			END_IF
		END_IF
	END_FOR
END_IF

(* Availability on a thirty second heartbeat, from whether ANY qualifying
   transaction succeeded in that window.

   Published every heartbeat while healthy, not only on change: that is how the
   rest of this project signals a device is alive - a last will on the PLC topic
   says it died, and a periodic online says it has not. *)
fbAvailTick(IN := NOT fbAvailTick.Q, PT := T#30S);

IF fbAvailTick.Q THEN
	IF uiTxSeen > 0 THEN
		bAvailable := uiTxOk > 0;
		bLastAvailable := bAvailable;
		bAvailabilityPublished := TRUE;
		THIS^.PubAvailability(Online := bAvailable);
	END_IF

	(* What the block actually saw, so the availability question can be settled
	   by looking rather than by reading source. txcalls counts every
	   OnTransactionDone; seen counts those with a required step; ok counts those
	   that succeeded; pubs counts availability messages this block sent. If pubs
	   is far below the number of offline messages on the broker, they are not
	   coming from here. *)
	sAvailDiag := CONCAT('txcalls=', UINT_TO_STRING(uiTxCalls));
	sAvailDiag := CONCAT(sAvailDiag, ' seen='); sAvailDiag := CONCAT(sAvailDiag, UINT_TO_STRING(uiTxSeen));
	sAvailDiag := CONCAT(sAvailDiag, ' ok='); sAvailDiag := CONCAT(sAvailDiag, UINT_TO_STRING(uiTxOk));
	sAvailDiag := CONCAT(sAvailDiag, ' pubs='); sAvailDiag := CONCAT(sAvailDiag, UINT_TO_STRING(uiAvailPubs));
	sAvailDiag := CONCAT(sAvailDiag, ' lastrun='); sAvailDiag := CONCAT(sAvailDiag, INT_TO_STRING(iLastStepsRun));
	sAvailDiag := CONCAT(sAvailDiag, ' lastfail='); sAvailDiag := CONCAT(sAvailDiag, INT_TO_STRING(iLastFailures));
	PubMqttMessage(Suffix := '/AVAIL_DIAG', Data := sAvailDiag);

	uiTxOk := 0;
	uiTxSeen := 0;
	uiTxCalls := 0;
END_IF


(* Every five minutes, publish the unit values again whether they moved or not,
   so a Home Assistant that reconnected still gets a value for a box that has
   been sitting in the same state. Matches the node blocks' own refresh. *)
fbMasterRefresh(IN := NOT fbMasterRefresh.Q, PT := T#5M);
IF fbMasterRefresh.Q THEN
	bRefreshDue := TRUE;

	(* The settings sweep runs again on the same clock, so a change made at the
	   box itself reaches Home Assistant without anybody touching it there. *)
	iBoxSettingsCursor := 0;
	bBoxSettingsDue := TRUE;
END_IF

          

METHOD InitRS485
  VAR_INPUT
    DataPollingInterval : TIME;
    DeviceAddress : BYTE;
  END_VAR
                  THIS^.fbTimerData.PT := DataPollingInterval;

THIS^.stMasterStep.DeviceId		:= DeviceAddress;
THIS^.stMasterStep.FunctionCode	:= 4;
THIS^.stMasterStep.Address		:= 10;
THIS^.stMasterStep.Quantity		:= 6;

(* Address and value are filled in by PublishReceived when a command arrives. *)
THIS^.stWriteStep.DeviceId		:= DeviceAddress;
THIS^.stWriteStep.FunctionCode	:= 6;
THIS^.stWriteStep.Quantity		:= 1;

THIS^.fbTimerData.IN := TRUE;

(* Same device, same holding registers as the write path uses. *)
THIS^.stBoxSettingsStep.DeviceId		:= DeviceAddress;
THIS^.stBoxSettingsStep.FunctionCode	:= 3;
THIS^.stBoxSettingsStep.Quantity		:= 1;

THIS^.bInitRS485Done := TRUE;

                
END_METHOD

METHOD InitMqtt
  VAR_INPUT
    MQTTPublishPrefix : POINTER TO STRING;
    MQTTSubscribePrefix : POINTER TO STRING;
    pMqttPublishQueue : POINTER TO FB_MQTT_PUBLISH_QUEUE;
    pMqttCallbackCollector : POINTER TO MQTT.CallbackCollector;
  END_VAR
                  SUPER^._sInstancePath := THIS^.sInstancePath; // Due to reflection its location is important

(*pass trough*)
THIS^.pMqttPublishQueue := pMqttPublishQueue;
THIS^.psMqttPublishTopicPrefix := MQTTPublishPrefix;
THIS^.psMqttSubscribeTopicPrefix := MQTTSubscribePrefix;
SUPER^.InitBaseMqtt();

// register the FB agains the collector so mqtt events can be received
pMqttCallbackCollector^.put(instance:= THIS^);


FOR iLoopCounter := 2 TO 30 DO
		afbNodes[iLoopCounter].InitMqtt(
			MQTTPublishPrefix := MQTTPublishPrefix,
			MqttPublishTopicSuffix := THIS^.MqttPublishTopicSuffix,
			pMqttPublishQueue := pMqttPublishQueue
		);
END_FOR
                
END_METHOD

METHOD PubMqttMessage
  VAR_INPUT
    Suffix : STRING(100);
    Data : STRING(100);
  END_VAR
                  IF bInitMqttDone THEN
		pMqttPublishQueue^.AddMessageOn(Lane := GVL_MQTT.MQTT_LANE_RS485,
			Payload := Data,
			Topic := CONCAT(THIS^.sMQTTPublishTopic, Suffix),
			Qos := MQTT.QoS.ExactlyOnce,
			MqttRetain := FALSE
		);
END_IF
                
END_METHOD

